Yaskawa INFORM job: DEMO_ROOF_SIDE_0625_3PAINT_53.JBI

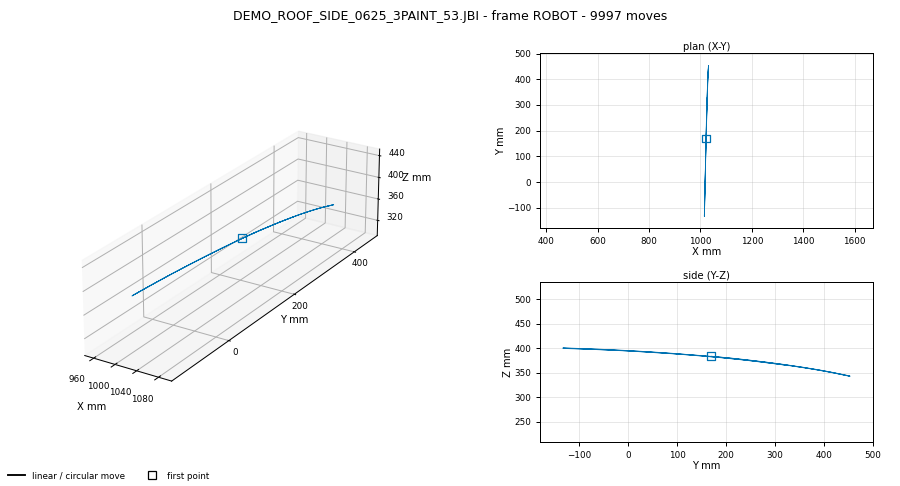
[picture p0: tool path of DEMO_ROOF_SIDE_0625_3PAINT_53.JBI in frame ROBOT, 9997 of 9997 moves have a stored position in this frame; points joined in program order, loops and branches not executed]
/JOB
//NAME DEMO_ROOF_SIDE_0625_3PAINT53
//POS
///NPOS 9997,0,0,0,0,0
///TOOL 0
///USER 0
///POSTYPE ROBOT
///RECTAN
///RCONF 1,0,0,0,0,0,0,0,0,0,0,0,0,0,0,0,0,0,0,0,0,0,0,0
C00000=1022.452,169.622,383.703,168.258,49.350,159.238
C00001=1022.457,169.870,383.681,168.261,49.345,159.237
C00002=1022.464,170.119,383.659,168.265,49.339,159.236
C00003=1022.469,170.368,383.637,168.268,49.333,159.236
C00004=1022.474,170.617,383.615,168.272,49.327,159.235
C00005=1022.480,170.866,383.593,168.276,49.321,159.234
C00006=1022.485,171.115,383.571,168.279,49.316,159.234
C00007=1022.491,171.398,383.546,168.283,49.310,159.233
C00008=1022.498,171.680,383.520,168.287,49.303,159.233
C00009=1022.504,171.963,383.496,168.291,49.296,159.232
C00010=1022.510,172.244,383.471,168.295,49.290,159.231
C00011=1022.515,172.494,383.449,168.299,49.284,159.231
C00012=1022.521,172.743,383.427,168.302,49.279,159.230
C00013=1022.526,172.991,383.404,168.306,49.273,159.229
C00014=1022.532,173.241,383.382,168.310,49.267,159.229
C00015=1022.537,173.489,383.361,168.313,49.261,159.228
C00016=1022.543,173.739,383.339,168.317,49.256,159.228
C00017=1022.548,173.988,383.316,168.320,49.250,159.227
C00018=1022.554,174.236,383.294,168.324,49.244,159.226
C00019=1022.559,174.486,383.272,168.328,49.238,159.226
C00020=1022.565,174.735,383.249,168.331,49.233,159.225
C00021=1022.571,174.983,383.228,168.335,49.227,159.225
C00022=1022.576,175.232,383.205,168.338,49.222,159.224
C00023=1022.582,175.481,383.183,168.342,49.216,159.223
C00024=1022.587,175.730,383.162,168.346,49.210,159.223
C00025=1022.593,175.979,383.139,168.349,49.204,159.222
C00026=1022.599,176.228,383.116,168.353,49.198,159.222
C00027=1022.603,176.477,383.094,168.357,49.193,159.221
C00028=1022.610,176.726,383.072,168.360,49.187,159.220
C00029=1022.615,176.975,383.050,168.364,49.181,159.220
C00030=1022.620,177.223,383.027,168.368,49.176,159.219
C00031=1022.627,177.473,383.006,168.372,49.170,159.219
C00032=1022.632,177.722,382.983,168.376,49.164,159.218
C00033=1022.637,177.970,382.961,168.379,49.159,159.217
C00034=1022.644,178.219,382.939,168.383,49.153,159.217
C00035=1022.649,178.469,382.916,168.387,49.147,159.216
C00036=1022.655,178.717,382.893,168.390,49.141,159.216
C00037=1022.660,178.966,382.871,168.394,49.136,159.215
C00038=1022.666,179.215,382.849,168.398,49.130,159.214
C00039=1022.671,179.464,382.827,168.401,49.125,159.214
C00040=1022.677,179.713,382.804,168.405,49.119,159.213
C00041=1022.683,179.962,382.783,168.409,49.113,159.213
C00042=1022.688,180.211,382.760,168.413,49.107,159.212
C00043=1022.694,180.460,382.738,168.416,49.102,159.211
C00044=1022.700,180.709,382.715,168.420,49.096,159.211
C00045=1022.706,180.958,382.693,168.424,49.090,159.210
C00046=1022.711,181.206,382.670,168.427,49.084,159.210
C00047=1022.717,181.455,382.647,168.432,49.079,159.209
C00048=1022.723,181.705,382.626,168.436,49.073,159.209
C00049=1022.729,181.953,382.603,168.440,49.067,159.208
C00050=1022.734,182.203,382.581,168.443,49.062,159.207
C00051=1022.740,182.452,382.558,168.447,49.056,159.207
C00052=1022.745,182.700,382.535,168.451,49.051,159.206
C00053=1022.750,182.949,382.512,168.454,49.045,159.206
C00054=1022.756,183.198,382.489,168.459,49.040,159.205
C00055=1022.761,183.448,382.466,168.462,49.034,159.205
C00056=1022.766,183.697,382.443,168.466,49.028,159.204
C00057=1022.771,183.945,382.420,168.470,49.023,159.204
C00058=1022.777,184.194,382.397,168.473,49.018,159.203
C00059=1022.782,184.443,382.374,168.478,49.013,159.203
C00060=1022.788,184.692,382.351,168.481,49.007,159.202
C00061=1022.793,184.941,382.328,168.485,49.002,159.201
C00062=1022.798,185.189,382.305,168.489,48.996,159.201
C00063=1022.803,185.438,382.282,168.492,48.991,159.200
C00064=1022.809,185.687,382.259,168.496,48.985,159.200
C00065=1022.814,185.936,382.235,168.501,48.980,159.199
C00066=1022.820,186.185,382.212,168.504,48.974,159.199
C00067=1022.826,186.434,382.189,168.508,48.969,159.198
C00068=1022.830,186.683,382.166,168.511,48.964,159.198
C00069=1022.836,186.932,382.143,168.515,48.958,159.197
C00070=1022.841,187.181,382.120,168.520,48.953,159.197
C00071=1022.848,187.462,382.094,168.524,48.947,159.196
C00072=1022.854,187.744,382.068,168.528,48.940,159.195
C00073=1022.860,188.026,382.041,168.532,48.934,159.195
C00074=1022.866,188.309,382.015,168.537,48.928,159.194
C00075=1022.871,188.558,381.992,168.541,48.922,159.194
C00076=1022.877,188.806,381.968,168.545,48.917,159.193
C00077=1022.882,189.055,381.945,168.549,48.911,159.193
C00078=1022.888,189.304,381.922,168.552,48.907,159.192
C00079=1022.894,189.553,381.899,168.556,48.901,159.191
C00080=1022.899,189.802,381.875,168.561,48.896,159.191
C00081=1022.905,190.051,381.852,168.564,48.890,159.190
C00082=1022.910,190.300,381.829,168.568,48.885,159.190
C00083=1022.916,190.548,381.805,168.572,48.879,159.189
C00084=1022.921,190.797,381.783,168.577,48.874,159.189
C00085=1022.926,191.046,381.759,168.580,48.868,159.188
C00086=1022.931,191.295,381.736,168.584,48.863,159.188
C00087=1022.937,191.543,381.712,168.588,48.857,159.187
C00088=1022.942,191.792,381.689,168.593,48.852,159.187
C00089=1022.948,192.041,381.666,168.596,48.847,159.186
C00090=1022.954,192.290,381.643,168.600,48.841,159.186
C00091=1022.959,192.539,381.619,168.604,48.836,159.185
C00092=1022.965,192.787,381.596,168.608,48.830,159.185
C00093=1022.971,193.036,381.573,168.611,48.825,159.184
C00094=1022.976,193.286,381.549,168.616,48.820,159.184
C00095=1022.982,193.534,381.526,168.620,48.814,159.183
C00096=1022.987,193.784,381.502,168.624,48.809,159.183
C00097=1022.993,194.033,381.479,168.628,48.803,159.182
C00098=1022.999,194.281,381.455,168.632,48.798,159.182
C00099=1023.004,194.530,381.432,168.636,48.792,159.181
C00100=1023.010,194.778,381.408,168.640,48.787,159.181
C00101=1023.016,195.027,381.385,168.644,48.781,159.180
C00102=1023.021,195.276,381.361,168.649,48.776,159.180
C00103=1023.027,195.525,381.338,168.653,48.770,159.179
C00104=1023.032,195.774,381.314,168.656,48.766,159.179
C00105=1023.038,196.023,381.291,168.660,48.760,159.178
C00106=1023.044,196.271,381.268,168.665,48.755,159.178
C00107=1023.049,196.520,381.244,168.669,48.749,159.177
C00108=1023.055,196.769,381.220,168.673,48.744,159.177
C00109=1023.061,197.018,381.197,168.677,48.738,159.176
C00110=1023.066,197.267,381.173,168.681,48.733,159.175
C00111=1023.072,197.516,381.150,168.685,48.727,159.175
C00112=1023.077,197.764,381.126,168.689,48.722,159.174
C00113=1023.083,198.013,381.103,168.693,48.716,159.174
C00114=1023.089,198.261,381.079,168.697,48.711,159.173
C00115=1023.095,198.511,381.055,168.702,48.706,159.173
C00116=1023.101,198.760,381.031,168.706,48.700,159.172
C00117=1023.106,199.009,381.008,168.710,48.695,159.172
C00118=1023.112,199.257,380.984,168.713,48.689,159.171
C00119=1023.117,199.506,380.961,168.718,48.684,159.171
C00120=1023.123,199.755,380.937,168.722,48.679,159.170
C00121=1023.129,200.004,380.913,168.726,48.673,159.170
C00122=1023.134,200.253,380.890,168.731,48.668,159.169
C00123=1023.140,200.501,380.865,168.735,48.663,159.169
C00124=1023.145,200.750,380.841,168.739,48.657,159.168
C00125=1023.151,200.999,380.816,168.743,48.653,159.168
C00126=1023.157,201.248,380.793,168.747,48.647,159.168
C00127=1023.162,201.497,380.769,168.751,48.642,159.167
C00128=1023.167,201.745,380.745,168.756,48.636,159.167
C00129=1023.173,201.994,380.721,168.760,48.631,159.166
C00130=1023.179,202.243,380.697,168.764,48.626,159.166
C00131=1023.184,202.492,380.672,168.769,48.621,159.165
C00132=1023.189,202.741,380.649,168.772,48.616,159.165
C00133=1023.195,202.989,380.625,168.776,48.610,159.164
C00134=1023.201,203.238,380.601,168.781,48.605,159.164
C00135=1023.225,204.270,380.500,169.200,48.703,159.246
C00136=1023.235,204.688,380.457,169.205,48.696,159.245
C00137=1023.246,205.107,380.414,169.211,48.689,159.244
C00138=1023.257,205.525,380.372,169.217,48.682,159.244
C00139=1023.268,205.943,380.328,169.222,48.674,159.243
C00140=1023.274,206.191,380.302,169.225,48.670,159.242
C00141=1023.281,206.440,380.277,169.228,48.666,159.242
C00142=1023.287,206.689,380.251,169.232,48.661,159.241
C00143=1023.294,206.937,380.225,169.234,48.657,159.241
C00144=1023.299,207.186,380.199,169.238,48.653,159.241
C00145=1023.306,207.434,380.173,169.241,48.648,159.240
C00146=1023.312,207.683,380.148,169.245,48.644,159.240
C00147=1023.319,207.932,380.121,169.248,48.640,159.239
C00148=1023.325,208.181,380.096,169.251,48.635,159.239
C00149=1023.332,208.429,380.070,169.255,48.631,159.238
C00150=1023.338,208.677,380.045,169.258,48.627,159.238
C00151=1023.345,208.926,380.018,169.261,48.623,159.238
C00152=1023.351,209.175,379.992,169.265,48.618,159.237
C00153=1023.357,209.423,379.966,169.267,48.615,159.237
C00154=1023.363,209.672,379.941,169.271,48.610,159.236
C00155=1023.371,209.920,379.914,169.275,48.606,159.236
C00156=1023.377,210.169,379.889,169.277,48.602,159.235
C00157=1023.383,210.417,379.862,169.281,48.598,159.235
C00158=1023.389,210.666,379.836,169.285,48.594,159.235
C00159=1023.396,210.915,379.811,169.287,48.590,159.234
C00160=1023.402,211.163,379.784,169.291,48.586,159.234
C00161=1023.408,211.411,379.758,169.295,48.581,159.234
C00162=1023.415,211.661,379.732,169.297,48.578,159.233
C00163=1023.421,211.909,379.706,169.301,48.573,159.233
C00164=1023.427,212.157,379.680,169.305,48.569,159.232
C00165=1023.433,212.406,379.654,169.307,48.565,159.232
C00166=1023.440,212.655,379.627,169.311,48.561,159.232
C00167=1023.446,212.903,379.601,169.315,48.557,159.231
C00168=1023.453,213.151,379.575,169.317,48.553,159.231
C00169=1023.459,213.401,379.549,169.321,48.549,159.230
C00170=1023.465,213.649,379.523,169.325,48.544,159.230
C00171=1023.471,213.897,379.496,169.327,48.541,159.230
C00172=1023.478,214.146,379.470,169.331,48.536,159.229
C00173=1023.485,214.394,379.444,169.335,48.532,159.229
C00174=1023.490,214.643,379.418,169.338,48.529,159.229
C00175=1023.497,214.892,379.391,169.341,48.524,159.228
C00176=1023.504,215.140,379.365,169.345,48.520,159.228
C00177=1023.510,215.389,379.339,169.348,48.516,159.227
C00178=1023.516,215.637,379.313,169.351,48.512,159.227
C00179=1023.523,215.885,379.287,169.355,48.508,159.227
C00180=1023.529,216.134,379.260,169.358,48.504,159.226
C00181=1023.536,216.382,379.234,169.362,48.500,159.226
C00182=1023.542,216.632,379.207,169.365,48.496,159.226
C00183=1023.549,216.880,379.181,169.368,48.492,159.225
C00184=1023.555,217.128,379.155,169.372,48.488,159.225
C00185=1023.561,217.377,379.128,169.375,48.484,159.224
C00186=1023.568,217.625,379.102,169.378,48.480,159.224
C00187=1023.575,217.874,379.076,169.382,48.476,159.224
C00188=1023.581,218.122,379.049,169.386,48.472,159.223
C00189=1023.587,218.371,379.023,169.388,48.468,159.223
C00190=1023.594,218.619,378.997,169.392,48.464,159.223
C00191=1023.600,218.868,378.970,169.396,48.460,159.222
C00192=1023.606,219.078,378.947,169.399,48.457,159.222
C00193=1023.611,219.289,378.925,169.401,48.454,159.222
C00194=1023.616,219.499,378.902,169.404,48.451,159.221
C00195=1023.622,219.710,378.879,169.407,48.447,159.221
C00196=1023.627,219.921,378.857,169.410,48.444,159.221
C00197=1023.632,220.131,378.834,169.413,48.441,159.221
C00198=1023.637,220.341,378.812,169.416,48.437,159.220
C00199=1023.643,220.552,378.789,169.419,48.434,159.220
C00200=1023.650,220.800,378.763,169.422,48.430,159.220
C00201=1023.656,221.049,378.736,169.425,48.426,159.219
C00202=1023.662,221.297,378.709,169.429,48.422,159.219
C00203=1023.669,221.546,378.683,169.432,48.419,159.219
C00204=1023.675,221.795,378.656,169.436,48.415,159.218
C00205=1023.681,222.044,378.629,169.439,48.411,159.218
C00206=1023.688,222.291,378.602,169.442,48.408,159.218
C00207=1023.694,222.540,378.575,169.446,48.404,159.217
C00208=1023.700,222.788,378.548,169.450,48.399,159.217
C00209=1023.707,223.037,378.522,169.453,48.396,159.217
C00210=1023.713,223.286,378.495,169.457,48.392,159.216
C00211=1023.719,223.534,378.468,169.459,48.388,159.216
C00212=1023.726,223.782,378.442,169.463,48.384,159.216
C00213=1023.732,224.031,378.415,169.467,48.381,159.215
C00214=1023.738,224.279,378.388,169.470,48.377,159.215
C00215=1023.746,224.528,378.361,169.474,48.373,159.215
C00216=1023.751,224.776,378.334,169.478,48.369,159.215
C00217=1023.758,225.025,378.307,169.480,48.366,159.214
C00218=1023.765,225.274,378.281,169.484,48.362,159.214
C00219=1023.771,225.522,378.253,169.488,48.358,159.214
C00220=1023.777,225.771,378.226,169.491,48.354,159.213
C00221=1023.784,226.019,378.200,169.495,48.351,159.213
C00222=1023.790,226.267,378.173,169.499,48.347,159.213
C00223=1023.797,226.516,378.146,169.501,48.343,159.212
C00224=1023.803,226.764,378.120,169.505,48.339,159.212
C00225=1023.810,227.013,378.092,169.508,48.336,159.212
C00226=1023.816,227.261,378.065,169.512,48.332,159.211
C00227=1023.822,227.509,378.037,169.516,48.328,159.211
C00228=1023.828,227.758,378.011,169.519,48.325,159.211
C00229=1023.835,228.007,377.984,169.523,48.321,159.210
C00230=1023.842,228.255,377.957,169.526,48.318,159.210
C00231=1023.848,228.503,377.930,169.530,48.314,159.210
C00232=1023.855,228.752,377.902,169.534,48.310,159.210
C00233=1023.861,229.001,377.875,169.537,48.307,159.209
C00234=1023.867,229.249,377.848,169.540,48.303,159.209
C00235=1023.874,229.497,377.820,169.544,48.299,159.209
C00236=1023.879,229.745,377.793,169.547,48.296,159.209
C00237=1023.886,229.994,377.766,169.551,48.292,159.208
C00238=1023.892,230.243,377.739,169.554,48.289,159.208
C00239=1023.899,230.491,377.711,169.558,48.285,159.208
C00240=1023.905,230.740,377.684,169.562,48.282,159.208
C00241=1023.912,230.988,377.657,169.565,48.278,159.207
C00242=1023.918,231.236,377.629,169.569,48.274,159.207
C00243=1023.924,231.485,377.602,169.572,48.271,159.207
C00244=1023.931,231.733,377.575,169.576,48.268,159.207
C00245=1023.937,231.981,377.547,169.580,48.264,159.206
C00246=1023.943,232.230,377.520,169.583,48.260,159.206
C00247=1023.950,232.479,377.492,169.587,48.257,159.206
C00248=1023.956,232.726,377.465,169.590,48.254,159.206
C00249=1023.963,232.975,377.437,169.594,48.250,159.205
C00250=1023.969,233.224,377.410,169.597,48.247,159.205
C00251=1023.975,233.473,377.382,169.601,48.243,159.205
C00252=1023.986,233.885,377.337,169.607,48.238,159.204
C00253=1023.997,234.298,377.291,169.612,48.232,159.204
C00254=1024.007,234.712,377.245,169.619,48.226,159.204
C00255=1024.017,235.125,377.199,169.625,48.220,159.203
C00256=1024.024,235.373,377.172,169.628,48.217,159.203
C00257=1024.031,235.621,377.144,169.632,48.213,159.203
C00258=1024.037,235.870,377.116,169.636,48.210,159.202
C00259=1024.043,236.118,377.089,169.639,48.207,159.202
C00260=1024.050,236.367,377.062,169.643,48.203,159.202
C00261=1024.056,236.615,377.034,169.646,48.199,159.202
C00262=1024.063,236.864,377.006,169.650,48.196,159.201
C00263=1024.069,237.112,376.978,169.654,48.193,159.201
C00264=1024.075,237.360,376.951,169.657,48.189,159.201
C00265=1024.082,237.609,376.923,169.661,48.186,159.201
C00266=1024.088,237.857,376.895,169.664,48.183,159.201
C00267=1024.095,238.105,376.868,169.668,48.179,159.200
C00268=1024.102,238.354,376.840,169.672,48.176,159.200
C00269=1024.108,238.603,376.811,169.675,48.173,159.200
C00270=1024.114,238.850,376.784,169.679,48.169,159.200
C00271=1024.120,239.099,376.756,169.684,48.166,159.200
C00272=1024.127,239.347,376.729,169.686,48.162,159.199
C00273=1024.134,239.596,376.701,169.690,48.159,159.199
C00274=1024.141,239.844,376.673,169.693,48.156,159.199
C00275=1024.146,240.092,376.645,169.698,48.153,159.199
C00276=1024.153,240.341,376.617,169.701,48.150,159.199
C00277=1024.158,240.589,376.589,169.705,48.146,159.198
C00278=1024.165,240.837,376.561,169.709,48.143,159.198
C00279=1024.171,241.086,376.532,169.712,48.140,159.198
C00280=1024.178,241.334,376.505,169.716,48.136,159.198
C00281=1024.185,241.583,376.477,169.719,48.133,159.198
C00282=1024.190,241.831,376.449,169.723,48.130,159.197
C00283=1024.197,242.079,376.421,169.727,48.126,159.197
C00284=1024.203,242.327,376.392,169.731,48.124,159.197
C00285=1024.210,242.576,376.364,169.735,48.121,159.197
C00286=1024.216,242.824,376.337,169.738,48.117,159.197
C00287=1024.223,243.072,376.308,169.742,48.114,159.197
C00288=1024.229,243.321,376.280,169.745,48.111,159.196
C00289=1024.235,243.570,376.252,169.749,48.107,159.196
C00290=1024.242,243.817,376.223,169.753,48.105,159.196
C00291=1024.248,244.065,376.195,169.757,48.102,159.196
C00292=1024.254,244.314,376.167,169.761,48.098,159.196
C00293=1024.261,244.562,376.138,169.764,48.095,159.195
C00294=1024.266,244.811,376.110,169.768,48.092,159.195
C00295=1024.273,245.059,376.081,169.771,48.089,159.195
C00296=1024.279,245.307,376.053,169.775,48.086,159.195
C00297=1024.286,245.556,376.024,169.779,48.083,159.195
C00298=1024.292,245.804,375.996,169.783,48.080,159.195
C00299=1024.299,246.052,375.968,169.787,48.077,159.195
C00300=1024.305,246.301,375.939,169.790,48.074,159.195
C00301=1024.311,246.549,375.910,169.794,48.071,159.194
C00302=1024.317,246.798,375.882,169.798,48.068,159.194
C00303=1024.324,247.046,375.853,169.802,48.065,159.194
C00304=1024.330,247.294,375.825,169.805,48.062,159.194
C00305=1024.336,247.542,375.796,169.809,48.059,159.194
C00306=1024.343,247.791,375.768,169.812,48.056,159.194
C00307=1024.349,248.039,375.739,169.817,48.053,159.194
C00308=1024.359,248.446,375.693,169.823,48.047,159.193
C00309=1024.370,248.853,375.646,169.829,48.043,159.193
C00310=1024.380,249.260,375.599,169.836,48.038,159.193
C00311=1024.390,249.666,375.551,169.841,48.033,159.193
C00312=1024.397,249.915,375.524,169.845,48.030,159.193
C00313=1024.403,250.163,375.495,169.849,48.027,159.192
C00314=1024.409,250.411,375.466,169.853,48.024,159.192
C00315=1024.416,250.660,375.438,169.856,48.021,159.192
C00316=1024.422,250.908,375.409,169.860,48.018,159.192
C00317=1024.429,251.156,375.380,169.865,48.015,159.192
C00318=1024.435,251.404,375.351,169.868,48.012,159.192
C00319=1024.442,251.652,375.323,169.872,48.009,159.192
C00320=1024.448,251.901,375.294,169.875,48.006,159.192
C00321=1024.454,252.149,375.265,169.880,48.004,159.192
C00322=1024.461,252.396,375.236,169.884,48.000,159.191
C00323=1024.468,252.646,375.208,169.887,47.998,159.191
C00324=1024.474,252.894,375.179,169.892,47.995,159.191
C00325=1024.480,253.142,375.150,169.895,47.992,159.191
C00326=1024.487,253.390,375.121,169.899,47.989,159.191
C00327=1024.493,253.638,375.092,169.903,47.986,159.191
C00328=1024.499,253.887,375.064,169.907,47.983,159.191
C00329=1024.506,254.135,375.035,169.911,47.980,159.191
C00330=1024.513,254.384,375.006,169.914,47.977,159.191
C00331=1024.519,254.632,374.977,169.918,47.975,159.191
C00332=1024.526,254.880,374.948,169.922,47.971,159.190
C00333=1024.533,255.128,374.920,169.926,47.969,159.190
C00334=1024.539,255.376,374.890,169.930,47.966,159.190
C00335=1024.546,255.625,374.861,169.934,47.963,159.190
C00336=1024.552,255.873,374.833,169.938,47.960,159.190
C00337=1024.559,256.121,374.804,169.942,47.957,159.190
C00338=1024.565,256.369,374.775,169.945,47.954,159.190
C00339=1024.571,256.617,374.746,169.950,47.952,159.190
C00340=1024.578,256.866,374.717,169.954,47.948,159.190
C00341=1024.585,257.114,374.688,169.957,47.946,159.189
C00342=1024.591,257.362,374.659,169.961,47.943,159.190
C00343=1024.597,257.610,374.630,169.966,47.940,159.190
C00344=1024.604,257.859,374.601,169.969,47.937,159.189
C00345=1024.611,258.107,374.572,169.973,47.934,159.189
C00346=1024.618,258.355,374.543,169.978,47.932,159.189
C00347=1024.624,258.604,374.514,169.981,47.929,159.189
C00348=1024.631,258.852,374.485,169.985,47.926,159.189
C00349=1024.638,259.100,374.456,169.990,47.923,159.189
C00350=1024.645,259.348,374.426,169.993,47.921,159.189
C00351=1024.651,259.596,374.397,169.997,47.917,159.189
C00352=1024.657,259.844,374.368,170.001,47.915,159.189
C00353=1024.665,260.093,374.339,170.005,47.912,159.189
C00354=1024.671,260.341,374.310,170.009,47.909,159.189
C00355=1024.677,260.589,374.281,170.014,47.907,159.189
C00356=1024.684,260.837,374.252,170.017,47.904,159.189
C00357=1024.691,261.086,374.222,170.022,47.901,159.189
C00358=1024.697,261.334,374.193,170.025,47.899,159.188
C00359=1024.703,261.582,374.164,170.029,47.896,159.188
C00360=1024.710,261.830,374.134,170.034,47.894,159.188
C00361=1024.716,262.078,374.104,170.037,47.891,159.188
C00362=1024.722,262.326,374.075,170.042,47.888,159.188
C00363=1024.729,262.575,374.045,170.045,47.886,159.188
C00364=1024.739,262.980,373.997,170.052,47.881,159.188
C00365=1024.750,263.385,373.948,170.058,47.877,159.188
C00366=1024.760,263.791,373.901,170.065,47.873,159.188
C00367=1024.772,264.196,373.852,170.072,47.869,159.188
C00368=1024.778,264.444,373.823,170.075,47.866,159.188
C00369=1024.785,264.692,373.793,170.080,47.863,159.188
C00370=1024.791,264.941,373.764,170.083,47.861,159.188
C00371=1024.798,265.189,373.733,170.088,47.858,159.188
C00372=1024.804,265.437,373.704,170.092,47.856,159.188
C00373=1024.811,265.684,373.675,170.095,47.853,159.188
C00374=1024.817,265.934,373.645,170.100,47.851,159.188
C00375=1024.824,266.181,373.615,170.105,47.848,159.188
C00376=1024.831,266.429,373.585,170.108,47.846,159.188
C00377=1024.836,266.678,373.555,170.112,47.843,159.188
C00378=1024.843,266.925,373.525,170.116,47.841,159.188
C00379=1024.850,267.173,373.495,170.120,47.839,159.188
C00380=1024.856,267.422,373.466,170.125,47.836,159.188
C00381=1024.863,267.670,373.435,170.128,47.833,159.188
C00382=1024.869,267.918,373.406,170.133,47.831,159.188
C00383=1024.876,268.166,373.376,170.137,47.829,159.188
C00384=1024.882,268.414,373.346,170.141,47.826,159.188
C00385=1024.889,268.662,373.316,170.145,47.823,159.188
C00386=1024.896,268.910,373.286,170.149,47.821,159.188
C00387=1024.902,269.159,373.256,170.153,47.819,159.188
C00388=1024.908,269.407,373.226,170.158,47.816,159.188
C00389=1024.915,269.655,373.196,170.161,47.814,159.188
C00390=1024.921,269.903,373.166,170.166,47.812,159.188
C00391=1024.928,270.151,373.136,170.170,47.809,159.188
C00392=1024.934,270.399,373.105,170.174,47.806,159.188
C00393=1024.941,270.647,373.075,170.178,47.804,159.188
C00394=1024.947,270.895,373.045,170.183,47.802,159.188
C00395=1024.954,271.144,373.015,170.186,47.800,159.189
C00396=1024.960,271.391,372.985,170.191,47.797,159.189
C00397=1024.967,271.640,372.955,170.195,47.795,159.189
C00398=1024.974,271.887,372.925,170.199,47.793,159.189
C00399=1024.980,272.136,372.895,170.204,47.791,159.189
C00400=1024.987,272.384,372.864,170.207,47.788,159.189
C00401=1024.993,272.632,372.834,170.212,47.785,159.189
C00402=1025.000,272.880,372.804,170.216,47.783,159.189
C00403=1025.006,273.128,372.774,170.220,47.781,159.189
C00404=1025.013,273.376,372.743,170.224,47.779,159.189
C00405=1025.020,273.624,372.712,170.229,47.777,159.189
C00406=1025.026,273.872,372.682,170.233,47.774,159.189
C00407=1025.033,274.120,372.652,170.237,47.772,159.189
C00408=1025.039,274.368,372.621,170.242,47.770,159.189
C00409=1025.046,274.616,372.591,170.245,47.768,159.189
C00410=1025.052,274.864,372.560,170.250,47.765,159.189
C00411=1025.058,275.112,372.530,170.255,47.763,159.189
C00412=1025.065,275.360,372.500,170.258,47.761,159.190
C00413=1025.072,275.608,372.468,170.263,47.758,159.190
C00414=1025.078,275.856,372.439,170.267,47.756,159.190
C00415=1025.085,276.104,372.408,170.271,47.754,159.190
C00416=1025.092,276.353,372.378,170.275,47.752,159.190
C00417=1025.098,276.600,372.347,170.280,47.750,159.190
C00418=1025.104,276.848,372.316,170.284,47.747,159.190
C00419=1025.112,277.097,372.286,170.288,47.745,159.190
C00420=1025.122,277.507,372.235,170.296,47.742,159.190
C00421=1025.132,277.916,372.184,170.302,47.738,159.190
C00422=1025.143,278.326,372.133,170.310,47.735,159.191
C00423=1025.154,278.736,372.083,170.317,47.731,159.191
C00424=1025.161,278.984,372.052,170.321,47.729,159.191
C00425=1025.168,279.232,372.020,170.326,47.727,159.191
C00426=1025.174,279.481,371.990,170.330,47.725,159.191
C00427=1025.180,279.728,371.959,170.334,47.723,159.191
C00428=1025.187,279.977,371.928,170.338,47.721,159.191
C00429=1025.194,280.224,371.897,170.343,47.719,159.192
C00430=1025.200,280.473,371.866,170.347,47.717,159.192
C00431=1025.207,280.720,371.835,170.352,47.715,159.192
C00432=1025.213,280.968,371.805,170.356,47.713,159.192
C00433=1025.220,281.216,371.773,170.360,47.711,159.192
C00434=1025.226,281.464,371.742,170.365,47.709,159.192
C00435=1025.234,281.712,371.712,170.369,47.706,159.192
C00436=1025.240,281.960,371.681,170.373,47.704,159.192
C00437=1025.246,282.208,371.650,170.378,47.702,159.193
C00438=1025.253,282.456,371.618,170.382,47.700,159.193
C00439=1025.260,282.704,371.587,170.387,47.698,159.193
C00440=1025.266,282.952,371.556,170.391,47.696,159.193
C00441=1025.273,283.200,371.525,170.395,47.694,159.193
C00442=1025.280,283.447,371.494,170.400,47.692,159.193
C00443=1025.286,283.696,371.464,170.404,47.691,159.193
C00444=1025.293,283.944,371.432,170.409,47.688,159.194
C00445=1025.299,284.192,371.401,170.413,47.686,159.194
C00446=1025.306,284.439,371.369,170.418,47.684,159.194
C00447=1025.313,284.688,371.339,170.422,47.683,159.194
C00448=1025.320,284.936,371.308,170.427,47.680,159.194
C00449=1025.327,285.183,371.276,170.431,47.678,159.194
C00450=1025.333,285.431,371.245,170.435,47.677,159.194
C00451=1025.340,285.679,371.213,170.440,47.675,159.195
C00452=1025.346,285.926,371.182,170.445,47.673,159.195
C00453=1025.353,286.174,371.151,170.449,47.671,159.195
C00454=1025.359,286.423,371.120,170.453,47.669,159.195
C00455=1025.366,286.671,371.089,170.458,47.667,159.195
C00456=1025.373,286.919,371.057,170.463,47.665,159.196
C00457=1025.379,287.167,371.025,170.467,47.664,159.196
C00458=1025.386,287.415,370.994,170.471,47.662,159.196
C00459=1025.392,287.663,370.962,170.476,47.660,159.196
C00460=1025.399,287.911,370.931,170.481,47.658,159.196
C00461=1025.406,288.159,370.900,170.485,47.657,159.197
C00462=1025.413,288.406,370.867,170.490,47.655,159.197
C00463=1025.420,288.654,370.836,170.494,47.653,159.197
C00464=1025.426,288.902,370.805,170.498,47.651,159.197
C00465=1025.433,289.150,370.773,170.503,47.649,159.197
C00466=1025.439,289.398,370.741,170.508,47.647,159.198
C00467=1025.446,289.646,370.710,170.513,47.645,159.198
C00468=1025.452,289.894,370.678,170.517,47.644,159.198
C00469=1025.459,290.141,370.647,170.521,47.642,159.198
C00470=1025.466,290.389,370.615,170.526,47.640,159.198
C00471=1025.473,290.637,370.583,170.531,47.638,159.199
C00472=1025.479,290.885,370.551,170.535,47.637,159.199
C00473=1025.486,291.133,370.520,170.540,47.635,159.199
C00474=1025.493,291.380,370.488,170.545,47.633,159.199
C00475=1025.500,291.629,370.456,170.549,47.631,159.199
C00476=1025.505,291.839,370.429,170.553,47.630,159.200
C00477=1025.511,292.051,370.402,170.557,47.628,159.200
C00478=1025.516,292.261,370.375,170.561,47.627,159.200
C00479=1025.523,292.472,370.348,170.565,47.626,159.200
C00480=1025.528,292.684,370.321,170.569,47.624,159.200
C00481=1025.533,292.895,370.293,170.573,47.623,159.201
C00482=1025.540,293.106,370.266,170.577,47.621,159.201
C00483=1025.545,293.317,370.238,170.581,47.620,159.201
C00484=1025.552,293.565,370.207,170.585,47.618,159.201
C00485=1025.559,293.813,370.175,170.590,47.617,159.202
C00486=1025.565,294.061,370.143,170.594,47.615,159.202
C00487=1025.572,294.308,370.111,170.599,47.613,159.202
C00488=1025.578,294.556,370.079,170.604,47.612,159.202
C00489=1025.585,294.804,370.046,170.609,47.611,159.203
C00490=1025.592,295.051,370.014,170.613,47.609,159.203
C00491=1025.598,295.300,369.981,170.618,47.607,159.203
C00492=1025.604,295.548,369.948,170.623,47.606,159.204
C00493=1025.611,295.795,369.916,170.627,47.605,159.204
C00494=1025.617,296.043,369.884,170.632,47.603,159.204
C00495=1025.624,296.290,369.852,170.637,47.601,159.204
C00496=1025.631,296.538,369.819,170.642,47.600,159.205
C00497=1025.637,296.787,369.787,170.646,47.599,159.205
C00498=1025.644,297.034,369.755,170.651,47.597,159.205
C00499=1025.651,297.282,369.722,170.656,47.595,159.206
C00500=1025.657,297.529,369.689,170.661,47.594,159.206
C00501=1025.664,297.777,369.657,170.666,47.592,159.206
C00502=1025.671,298.026,369.625,170.670,47.591,159.206
C00503=1025.677,298.273,369.592,170.675,47.590,159.207
C00504=1025.684,298.520,369.560,170.680,47.588,159.207
C00505=1025.690,298.768,369.527,170.685,47.586,159.207
C00506=1025.698,299.016,369.495,170.689,47.585,159.208
C00507=1025.704,299.264,369.462,170.694,47.584,159.208
C00508=1025.710,299.511,369.429,170.699,47.582,159.208
C00509=1025.717,299.759,369.398,170.704,47.581,159.209
C00510=1025.724,300.007,369.365,170.709,47.580,159.209
C00511=1025.730,300.255,369.332,170.713,47.578,159.209
C00512=1025.737,300.502,369.300,170.718,47.577,159.210
C00513=1025.744,300.751,369.267,170.723,47.576,159.210
C00514=1025.751,300.998,369.234,170.728,47.574,159.210
C00515=1025.758,301.245,369.202,170.733,47.573,159.211
C00516=1025.764,301.494,369.169,170.737,47.572,159.211
C00517=1025.771,301.741,369.136,170.742,47.570,159.211
C00518=1025.778,301.989,369.103,170.747,47.569,159.212
C00519=1025.785,302.236,369.070,170.752,47.567,159.212
C00520=1025.791,302.484,369.037,170.757,47.566,159.212
C00521=1025.799,302.732,369.005,170.762,47.564,159.213
C00522=1025.805,302.979,368.972,170.767,47.563,159.213
C00523=1025.812,303.228,368.939,170.771,47.562,159.213
C00524=1025.819,303.475,368.907,170.776,47.560,159.214
C00525=1025.825,303.723,368.874,170.781,47.559,159.214
C00526=1025.832,303.971,368.841,170.786,47.558,159.214
C00527=1025.840,304.218,368.808,170.791,47.556,159.215
C00528=1025.847,304.466,368.775,170.797,47.555,159.215
C00529=1025.853,304.713,368.742,170.802,47.554,159.215
C00530=1025.861,304.961,368.710,170.806,47.553,159.216
C00531=1025.867,305.208,368.676,170.811,47.551,159.216
C00532=1025.874,305.457,368.643,170.816,47.550,159.216
C00533=1025.881,305.704,368.611,170.821,47.549,159.217
C00534=1025.888,305.952,368.578,170.826,47.547,159.217
C00535=1025.895,306.200,368.544,170.831,47.546,159.218
C00536=1025.901,306.419,368.515,170.835,47.545,159.218
C00537=1025.907,306.639,368.486,170.840,47.544,159.218
C00538=1025.914,306.859,368.457,170.845,47.543,159.219
C00539=1025.920,307.078,368.427,170.849,47.542,159.219
C00540=1025.926,307.298,368.398,170.854,47.541,159.219
C00541=1025.933,307.518,368.368,170.858,47.540,159.220
C00542=1025.939,307.738,368.339,170.862,47.538,159.220
C00543=1025.945,307.958,368.310,170.867,47.537,159.220
C00544=1025.952,308.205,368.277,170.872,47.536,159.221
C00545=1025.959,308.453,368.243,170.877,47.535,159.221
C00546=1025.966,308.700,368.211,170.882,47.533,159.221
C00547=1025.973,308.948,368.177,170.888,47.533,159.222
C00548=1025.980,309.196,368.144,170.892,47.531,159.222
C00549=1025.987,309.443,368.111,170.897,47.530,159.223
C00550=1025.994,309.691,368.078,170.902,47.529,159.223
C00551=1026.001,309.939,368.044,170.907,47.528,159.223
C00552=1026.008,310.186,368.012,170.912,47.526,159.224
C00553=1026.016,310.434,367.979,170.918,47.526,159.224
C00554=1026.023,310.681,367.945,170.923,47.524,159.225
C00555=1026.029,310.929,367.912,170.928,47.523,159.225
C00556=1026.036,311.177,367.878,170.933,47.522,159.226
C00557=1026.043,311.425,367.844,170.938,47.521,159.226
C00558=1026.049,311.672,367.810,170.944,47.520,159.227
C00559=1026.057,311.919,367.776,170.949,47.519,159.227
C00560=1026.063,312.167,367.742,170.954,47.518,159.227
C00561=1026.070,312.414,367.709,170.959,47.518,159.228
C00562=1026.077,312.662,367.675,170.964,47.517,159.228
C00563=1026.083,312.910,367.640,170.969,47.515,159.229
C00564=1026.090,313.157,367.607,170.974,47.515,159.229
C00565=1026.097,313.405,367.573,170.980,47.514,159.230
C00566=1026.104,313.653,367.539,170.985,47.512,159.230
C00567=1026.111,313.900,367.505,170.990,47.512,159.231
C00568=1026.117,314.147,367.471,170.995,47.511,159.231
C00569=1026.125,314.395,367.437,171.001,47.510,159.232
C00570=1026.131,314.643,367.403,171.006,47.509,159.232
C00571=1026.138,314.891,367.369,171.011,47.508,159.233
C00572=1026.145,315.138,367.336,171.017,47.507,159.233
C00573=1026.152,315.385,367.301,171.022,47.506,159.234
C00574=1026.159,315.633,367.267,171.026,47.506,159.234
C00575=1026.166,315.880,367.233,171.032,47.505,159.235
C00576=1026.173,316.128,367.199,171.037,47.504,159.235
C00577=1026.180,316.376,367.165,171.042,47.503,159.236
C00578=1026.186,316.623,367.131,171.048,47.503,159.236
C00579=1026.193,316.870,367.096,171.053,47.501,159.236
C00580=1026.200,317.118,367.062,171.058,47.500,159.237
C00581=1026.208,317.366,367.029,171.063,47.500,159.238
C00582=1026.214,317.613,366.993,171.069,47.499,159.238
C00583=1026.221,317.861,366.960,171.074,47.498,159.239
C00584=1026.229,318.108,366.926,171.079,47.497,159.239
C00585=1026.235,318.356,366.891,171.085,47.496,159.240
C00586=1026.243,318.603,366.857,171.090,47.496,159.240
C00587=1026.250,318.851,366.823,171.096,47.495,159.241
C00588=1026.257,319.098,366.788,171.101,47.494,159.241
C00589=1026.264,319.346,366.754,171.106,47.493,159.242
C00590=1026.271,319.594,366.720,171.112,47.492,159.242
C00591=1026.278,319.841,366.685,171.117,47.492,159.243
C00592=1026.285,320.089,366.651,171.123,47.491,159.243
C00593=1026.293,320.336,366.617,171.129,47.490,159.244
C00594=1026.299,320.584,366.582,171.134,47.490,159.245
C00595=1026.306,320.831,366.548,171.140,47.489,159.245
C00596=1026.312,321.053,366.517,171.144,47.488,159.246
C00597=1026.319,321.276,366.486,171.149,47.487,159.246
C00598=1026.325,321.498,366.455,171.154,47.487,159.247
C00599=1026.332,321.720,366.425,171.159,47.486,159.247
C00600=1026.339,321.942,366.393,171.163,47.486,159.247
C00601=1026.345,322.164,366.362,171.169,47.485,159.248
C00602=1026.351,322.387,366.331,171.173,47.484,159.248
C00603=1026.358,322.609,366.300,171.178,47.484,159.249
C00604=1026.365,322.856,366.266,171.184,47.483,159.250
C00605=1026.371,323.104,366.231,171.189,47.483,159.250
C00606=1026.380,323.352,366.196,171.195,47.482,159.251
C00607=1026.387,323.599,366.162,171.200,47.481,159.251
C00608=1026.394,323.846,366.127,171.207,47.480,159.252
C00609=1026.401,324.094,366.093,171.212,47.480,159.253
C00610=1026.409,324.341,366.058,171.218,47.479,159.253
C00611=1026.416,324.589,366.023,171.223,47.479,159.254
C00612=1026.423,324.836,365.988,171.229,47.478,159.254
C00613=1026.430,325.084,365.954,171.234,47.477,159.255
C00614=1026.437,325.331,365.919,171.240,47.477,159.256
C00615=1026.446,325.579,365.884,171.245,47.476,159.256
C00616=1026.452,325.826,365.849,171.251,47.475,159.257
C00617=1026.460,326.073,365.815,171.257,47.475,159.257
C00618=1026.468,326.321,365.780,171.262,47.474,159.258
C00619=1026.475,326.568,365.745,171.268,47.474,159.259
C00620=1026.482,326.816,365.711,171.273,47.473,159.259
C00621=1026.489,327.064,365.675,171.279,47.472,159.260
C00622=1026.497,327.311,365.641,171.285,47.472,159.260
C00623=1026.504,327.558,365.605,171.291,47.472,159.261
C00624=1026.512,327.806,365.570,171.296,47.471,159.262
C00625=1026.519,328.053,365.535,171.302,47.471,159.262
C00626=1026.525,328.300,365.500,171.308,47.471,159.263
C00627=1026.532,328.548,365.465,171.313,47.470,159.264
C00628=1026.540,328.795,365.428,171.319,47.470,159.264
C00629=1026.547,329.042,365.394,171.325,47.469,159.265
C00630=1026.555,329.290,365.358,171.331,47.468,159.265
C00631=1026.562,329.538,365.323,171.336,47.468,159.266
C00632=1026.569,329.785,365.287,171.342,47.468,159.267
C00633=1026.576,330.033,365.252,171.348,47.468,159.268
C00634=1026.583,330.280,365.217,171.353,47.467,159.268
C00635=1026.591,330.527,365.181,171.360,47.466,159.269
C00636=1026.598,330.774,365.146,171.365,47.466,159.270
C00637=1026.605,331.022,365.111,171.371,47.466,159.270
C00638=1026.612,331.269,365.075,171.377,47.466,159.271
C00639=1026.619,331.517,365.039,171.382,47.466,159.272
C00640=1026.627,331.764,365.003,171.389,47.465,159.272
C00641=1026.634,332.011,364.969,171.394,47.464,159.273
C00642=1026.642,332.259,364.932,171.400,47.464,159.274
C00643=1026.649,332.506,364.897,171.406,47.464,159.274
C00644=1026.656,332.753,364.861,171.411,47.464,159.275
C00645=1026.663,333.001,364.826,171.418,47.463,159.276
C00646=1026.671,333.248,364.790,171.424,47.463,159.277
C00647=1026.679,333.496,364.755,171.430,47.463,159.277
C00648=1026.686,333.743,364.719,171.435,47.463,159.278
C00649=1026.694,333.990,364.683,171.442,47.462,159.279
C00650=1026.701,334.237,364.647,171.448,47.462,159.279
C00651=1026.708,334.485,364.611,171.453,47.462,159.280
C00652=1026.715,334.732,364.575,171.459,47.462,159.281
C00653=1026.722,334.979,364.539,171.466,47.461,159.282
C00654=1026.730,335.227,364.503,171.472,47.462,159.283
C00655=1026.737,335.474,364.467,171.477,47.462,159.283
C00656=1026.744,335.694,364.436,171.483,47.462,159.284
C00657=1026.750,335.914,364.403,171.488,47.462,159.285
C00658=1026.757,336.134,364.371,171.493,47.461,159.285
C00659=1026.763,336.354,364.339,171.499,47.461,159.286
C00660=1026.770,336.574,364.307,171.505,47.461,159.287
C00661=1026.776,336.794,364.275,171.509,47.461,159.287
C00662=1026.783,337.014,364.242,171.515,47.461,159.288
C00663=1026.790,337.234,364.210,171.520,47.461,159.289
C00664=1026.797,337.481,364.174,171.526,47.461,159.289
C00665=1026.804,337.729,364.138,171.532,47.460,159.290
C00666=1026.812,337.976,364.102,171.539,47.461,159.291
C00667=1026.820,338.224,364.065,171.544,47.460,159.292
C00668=1026.827,338.470,364.029,171.550,47.460,159.292
C00669=1026.834,338.718,363.993,171.557,47.460,159.293
C00670=1026.842,338.965,363.957,171.563,47.460,159.294
C00671=1026.850,339.213,363.921,171.568,47.460,159.295
C00672=1026.857,339.459,363.884,171.575,47.460,159.296
C00673=1026.865,339.706,363.848,171.581,47.460,159.297
C00674=1026.872,339.954,363.812,171.587,47.460,159.297
C00675=1026.879,340.201,363.775,171.594,47.460,159.298
C00676=1026.887,340.448,363.738,171.600,47.460,159.299
C00677=1026.895,340.696,363.702,171.605,47.460,159.300
C00678=1026.901,340.943,363.665,171.612,47.460,159.301
C00679=1026.909,341.190,363.628,171.618,47.460,159.301
C00680=1026.917,341.437,363.592,171.624,47.460,159.302
C00681=1026.924,341.685,363.555,171.631,47.461,159.303
C00682=1026.932,341.932,363.519,171.637,47.460,159.304
C00683=1026.940,342.179,363.482,171.643,47.461,159.305
C00684=1026.947,342.426,363.445,171.650,47.461,159.306
C00685=1026.955,342.674,363.409,171.655,47.461,159.307
C00686=1026.963,342.921,363.372,171.662,47.461,159.307
C00687=1026.969,343.168,363.335,171.668,47.461,159.308
C00688=1026.977,343.415,363.298,171.674,47.462,159.309
C00689=1026.984,343.662,363.261,171.681,47.461,159.310
C00690=1026.992,343.909,363.224,171.687,47.462,159.311
C00691=1027.000,344.156,363.188,171.694,47.462,159.312
C00692=1027.007,344.404,363.151,171.700,47.462,159.313
C00693=1027.015,344.650,363.114,171.707,47.462,159.314
C00694=1027.022,344.898,363.076,171.713,47.463,159.315
C00695=1027.030,345.145,363.039,171.719,47.463,159.315
C00696=1027.037,345.393,363.002,171.726,47.463,159.316
C00697=1027.045,345.640,362.965,171.732,47.463,159.317
C00698=1027.053,345.886,362.928,171.739,47.463,159.318
C00699=1027.061,346.134,362.891,171.745,47.464,159.319
C00700=1027.069,346.380,362.854,171.752,47.464,159.320
C00701=1027.076,346.628,362.816,171.758,47.464,159.321
C00702=1027.084,346.875,362.780,171.764,47.464,159.322
C00703=1027.091,347.122,362.743,171.770,47.465,159.323
C00704=1027.099,347.369,362.706,171.777,47.465,159.324
C00705=1027.107,347.617,362.668,171.783,47.465,159.325
C00706=1027.115,347.864,362.631,171.791,47.466,159.326
C00707=1027.122,348.111,362.593,171.797,47.466,159.327
C00708=1027.130,348.358,362.556,171.804,47.467,159.327
C00709=1027.137,348.605,362.519,171.810,47.467,159.328
C00710=1027.146,348.852,362.481,171.817,47.467,159.329
C00711=1027.153,349.099,362.443,171.823,47.468,159.330
C00712=1027.160,349.346,362.406,171.830,47.468,159.331
C00713=1027.168,349.593,362.369,171.836,47.469,159.332
C00714=1027.176,349.840,362.331,171.843,47.469,159.333
C00715=1027.184,350.087,362.293,171.849,47.470,159.334
C00716=1027.190,350.305,362.259,171.855,47.470,159.335
C00717=1027.197,350.524,362.227,171.861,47.470,159.336
C00718=1027.204,350.742,362.193,171.867,47.470,159.337
C00719=1027.211,350.961,362.160,171.873,47.471,159.338
C00720=1027.218,351.180,362.126,171.879,47.471,159.339
C00721=1027.225,351.397,362.093,171.885,47.472,159.339
C00722=1027.231,351.616,362.060,171.891,47.472,159.340
C00723=1027.238,351.834,362.026,171.897,47.473,159.341
C00724=1027.245,352.081,361.989,171.903,47.473,159.342
C00725=1027.254,352.328,361.951,171.910,47.474,159.343
C00726=1027.262,352.576,361.913,171.917,47.474,159.344
C00727=1027.270,352.823,361.875,171.923,47.475,159.345
C00728=1027.278,353.070,361.838,171.931,47.475,159.346
C00729=1027.285,353.316,361.799,171.938,47.476,159.348
C00730=1027.293,353.564,361.761,171.944,47.477,159.348
C00731=1027.301,353.810,361.723,171.951,47.477,159.350
C00732=1027.310,354.057,361.685,171.957,47.478,159.350
C00733=1027.317,354.304,361.648,171.965,47.478,159.352
C00734=1027.325,354.552,361.609,171.972,47.479,159.353
C00735=1027.333,354.798,361.571,171.978,47.480,159.354
C00736=1027.341,355.046,361.534,171.985,47.480,159.355
C00737=1027.349,355.292,361.495,171.993,47.481,159.356
C00738=1027.357,355.539,361.457,171.999,47.482,159.357
C00739=1027.364,355.786,361.418,172.006,47.482,159.358
C00740=1027.373,356.033,361.380,172.013,47.483,159.359
C00741=1027.380,356.280,361.342,172.020,47.484,159.360
C00742=1027.388,356.527,361.303,172.027,47.485,159.361
C00743=1027.396,356.773,361.265,172.034,47.485,159.362
C00744=1027.404,357.021,361.226,172.041,47.486,159.364
C00745=1027.412,357.268,361.187,172.048,47.487,159.365
C00746=1027.420,357.514,361.149,172.055,47.487,159.366
C00747=1027.428,357.762,361.111,172.062,47.488,159.367
C00748=1027.437,358.009,361.073,172.069,47.489,159.368
C00749=1027.444,358.255,361.034,172.076,47.490,159.369
C00750=1027.452,358.502,360.996,172.083,47.490,159.370
C00751=1027.461,358.749,360.957,172.090,47.491,159.371
C00752=1027.468,358.996,360.919,172.097,47.492,159.372
C00753=1027.477,359.243,360.880,172.104,47.493,159.374
C00754=1027.485,359.490,360.841,172.111,47.494,159.375
C00755=1027.492,359.736,360.803,172.119,47.495,159.376
C00756=1027.500,359.984,360.764,172.126,47.495,159.377
C00757=1027.509,360.230,360.725,172.133,47.496,159.378
C00758=1027.517,360.477,360.686,172.140,47.497,159.379
C00759=1027.525,360.724,360.648,172.147,47.498,159.381
C00760=1027.532,360.971,360.608,172.155,47.499,159.382
C00761=1027.540,361.218,360.569,172.162,47.500,159.383
C00762=1027.549,361.465,360.530,172.170,47.501,159.384
C00763=1027.557,361.712,360.491,172.177,47.502,159.385
C00764=1027.564,361.958,360.452,172.183,47.503,159.387
C00765=1027.573,362.205,360.413,172.191,47.504,159.388
C00766=1027.581,362.452,360.374,172.198,47.505,159.389
C00767=1027.589,362.698,360.335,172.206,47.506,159.390
C00768=1027.597,362.945,360.295,172.213,47.507,159.392
C00769=1027.605,363.193,360.256,172.221,47.508,159.393
C00770=1027.613,363.438,360.217,172.228,47.509,159.394
C00771=1027.621,363.685,360.178,172.235,47.510,159.395
C00772=1027.629,363.932,360.138,172.242,47.511,159.396
C00773=1027.637,364.179,360.099,172.250,47.512,159.398
C00774=1027.646,364.426,360.060,172.257,47.513,159.399
C00775=1027.654,364.672,360.021,172.264,47.514,159.400
C00776=1027.661,364.894,359.985,172.271,47.515,159.401
C00777=1027.669,365.116,359.949,172.278,47.516,159.402
C00778=1027.676,365.338,359.915,172.284,47.517,159.404
C00779=1027.683,365.559,359.879,172.291,47.519,159.405
C00780=1027.691,365.780,359.843,172.298,47.519,159.406
C00781=1027.699,366.003,359.808,172.305,47.520,159.407
C00782=1027.706,366.224,359.772,172.312,47.521,159.408
C00783=1027.713,366.446,359.737,172.319,47.523,159.409
C00784=1027.721,366.693,359.697,172.326,47.524,159.411
C00785=1027.730,366.940,359.658,172.334,47.525,159.412
C00786=1027.738,367.186,359.618,172.341,47.526,159.413
C00787=1027.747,367.433,359.578,172.349,47.527,159.415
C00788=1027.755,367.680,359.538,172.356,47.528,159.416
C00789=1027.764,367.926,359.499,172.364,47.530,159.417
C00790=1027.772,368.173,359.460,172.372,47.531,159.419
C00791=1027.780,368.420,359.420,172.379,47.532,159.420
C00792=1027.788,368.666,359.380,172.387,47.534,159.421
C00793=1027.798,368.913,359.340,172.395,47.535,159.423
C00794=1027.805,369.160,359.300,172.402,47.536,159.424
C00795=1027.814,369.406,359.260,172.410,47.537,159.425
C00796=1027.822,369.653,359.220,172.419,47.538,159.427
C00797=1027.831,369.899,359.180,172.426,47.540,159.428
C00798=1027.839,370.147,359.140,172.434,47.541,159.429
C00799=1027.847,370.393,359.099,172.442,47.543,159.431
C00800=1027.856,370.639,359.059,172.449,47.544,159.432
C00801=1027.863,370.886,359.019,172.457,47.545,159.434
C00802=1027.872,371.133,358.978,172.465,47.547,159.435
C00803=1027.881,371.379,358.938,172.473,47.548,159.436
C00804=1027.888,371.626,358.898,172.480,47.550,159.438
C00805=1027.898,371.872,358.858,172.489,47.551,159.439
C00806=1027.906,372.119,358.817,172.497,47.553,159.441
C00807=1027.914,372.365,358.777,172.504,47.554,159.442
C00808=1027.923,372.612,358.737,172.512,47.556,159.444
C00809=1027.931,372.858,358.696,172.520,47.557,159.445
C00810=1027.940,373.105,358.656,172.528,47.559,159.446
C00811=1027.948,373.351,358.615,172.537,47.560,159.448
C00812=1027.957,373.598,358.574,172.545,47.562,159.449
C00813=1027.966,373.844,358.534,172.552,47.563,159.451
C00814=1027.974,374.091,358.493,172.560,47.565,159.452
C00815=1027.983,374.337,358.453,172.569,47.566,159.454
C00816=1027.992,374.584,358.412,172.577,47.568,159.455
C00817=1028.000,374.831,358.371,172.585,47.570,159.457
C00818=1028.009,375.077,358.331,172.592,47.571,159.458
C00819=1028.017,375.324,358.290,172.601,47.572,159.460
C00820=1028.026,375.571,358.249,172.609,47.574,159.461
C00821=1028.035,375.816,358.209,172.617,47.576,159.463
C00822=1028.044,376.063,358.168,172.626,47.577,159.464
C00823=1028.053,376.310,358.127,172.634,47.579,159.466
C00824=1028.061,376.556,358.087,172.642,47.581,159.467
C00825=1028.070,376.803,358.046,172.651,47.582,159.469
C00826=1028.079,377.049,358.004,172.659,47.584,159.470
C00827=1028.087,377.295,357.964,172.667,47.586,159.472
C00828=1028.096,377.542,357.923,172.676,47.587,159.473
C00829=1028.105,377.788,357.881,172.684,47.589,159.475
C00830=1028.113,378.035,357.840,172.692,47.591,159.477
C00831=1028.122,378.281,357.799,172.701,47.593,159.478
C00832=1028.131,378.528,357.757,172.709,47.595,159.480
C00833=1028.139,378.774,357.716,172.717,47.596,159.481
C00834=1028.148,379.020,357.675,172.726,47.598,159.483
C00835=1028.157,379.267,357.633,172.733,47.600,159.484
C00836=1028.165,379.499,357.595,172.741,47.602,159.486
C00837=1028.173,379.731,357.555,172.749,47.603,159.487
C00838=1028.182,379.963,357.516,172.757,47.605,159.489
C00839=1028.189,380.195,357.477,172.765,47.607,159.491
C00840=1028.198,380.428,357.438,172.774,47.609,159.492
C00841=1028.206,380.661,357.399,172.782,47.610,159.494
C00842=1028.214,380.892,357.360,172.790,47.612,159.495
C00843=1028.223,381.125,357.320,172.798,47.614,159.497
C00844=1028.232,381.371,357.278,172.806,47.616,159.498
C00845=1028.241,381.618,357.237,172.816,47.618,159.500
C00846=1028.249,381.864,357.195,172.823,47.620,159.502
C00847=1028.258,382.110,357.153,172.833,47.622,159.503
C00848=1028.267,382.357,357.112,172.842,47.624,159.505
C00849=1028.276,382.603,357.070,172.850,47.626,159.507
C00850=1028.285,382.849,357.028,172.859,47.627,159.508
C00851=1028.294,383.096,356.986,172.867,47.630,159.510
C00852=1028.303,383.342,356.944,172.877,47.632,159.512
C00853=1028.313,383.588,356.903,172.885,47.634,159.513
C00854=1028.322,383.834,356.861,172.894,47.636,159.515
C00855=1028.331,384.080,356.819,172.903,47.638,159.517
C00856=1028.340,384.326,356.777,172.911,47.640,159.519
C00857=1028.349,384.572,356.735,172.920,47.642,159.520
C00858=1028.358,384.819,356.694,172.930,47.644,159.522
C00859=1028.367,385.065,356.651,172.938,47.646,159.524
C00860=1028.377,385.312,356.609,172.947,47.649,159.526
C00861=1028.386,385.558,356.567,172.957,47.651,159.527
C00862=1028.395,385.804,356.525,172.965,47.653,159.529
C00863=1028.404,386.050,356.483,172.974,47.655,159.531
C00864=1028.413,386.296,356.441,172.983,47.657,159.533
C00865=1028.423,386.542,356.398,172.993,47.659,159.534
C00866=1028.431,386.789,356.356,173.001,47.662,159.536
C00867=1028.440,387.035,356.313,173.010,47.664,159.538
C00868=1028.450,387.281,356.270,173.020,47.666,159.540
C00869=1028.459,387.527,356.228,173.029,47.668,159.542
C00870=1028.468,387.774,356.186,173.037,47.670,159.543
C00871=1028.477,388.019,356.143,173.047,47.672,159.545
C00872=1028.487,388.266,356.100,173.056,47.675,159.547
C00873=1028.496,388.511,356.058,173.066,47.677,159.549
C00874=1028.504,388.758,356.015,173.075,47.679,159.551
C00875=1028.514,389.004,355.972,173.084,47.682,159.553
C00876=1028.524,389.250,355.930,173.093,47.684,159.555
C00877=1028.533,389.496,355.887,173.102,47.686,159.556
C00878=1028.542,389.742,355.844,173.112,47.689,159.558
C00879=1028.552,389.989,355.801,173.121,47.691,159.560
C00880=1028.561,390.234,355.759,173.131,47.694,159.562
C00881=1028.570,390.480,355.715,173.140,47.696,159.564
C00882=1028.580,390.726,355.672,173.149,47.699,159.566
C00883=1028.589,390.973,355.629,173.158,47.701,159.568
C00884=1028.598,391.218,355.586,173.168,47.704,159.570
C00885=1028.608,391.465,355.543,173.177,47.706,159.572
C00886=1028.617,391.711,355.500,173.187,47.709,159.574
C00887=1028.627,391.957,355.456,173.197,47.711,159.576
C00888=1028.635,392.203,355.413,173.206,47.714,159.578
C00889=1028.645,392.448,355.370,173.215,47.716,159.580
C00890=1028.655,392.695,355.326,173.225,47.719,159.582
C00891=1028.664,392.940,355.283,173.235,47.721,159.584
C00892=1028.674,393.187,355.240,173.244,47.724,159.586
C00893=1028.683,393.433,355.196,173.254,47.727,159.588
C00894=1028.693,393.678,355.153,173.264,47.729,159.590
C00895=1028.702,393.925,355.110,173.273,47.732,159.592
C00896=1028.712,394.179,355.064,173.284,47.734,159.594
C00897=1028.722,394.433,355.019,173.294,47.738,159.596
C00898=1028.732,394.688,354.974,173.304,47.740,159.598
C00899=1028.742,394.943,354.928,173.315,47.743,159.600
C00900=1028.751,395.188,354.885,173.324,47.746,159.602
C00901=1028.761,395.434,354.841,173.334,47.748,159.604
C00902=1028.771,395.680,354.798,173.344,47.751,159.606
C00903=1028.780,395.926,354.754,173.354,47.754,159.608
C00904=1028.790,396.172,354.709,173.364,47.756,159.610
C00905=1028.800,396.418,354.666,173.374,47.759,159.612
C00906=1028.809,396.664,354.622,173.384,47.762,159.615
C00907=1028.819,396.909,354.579,173.393,47.765,159.617
C00908=1028.828,397.155,354.534,173.403,47.768,159.619
C00909=1028.838,397.401,354.490,173.414,47.770,159.621
C00910=1028.848,397.647,354.446,173.424,47.774,159.623
C00911=1028.858,397.892,354.401,173.434,47.776,159.625
C00912=1028.868,398.138,354.358,173.444,47.779,159.627
C00913=1028.877,398.384,354.314,173.455,47.782,159.630
C00914=1028.887,398.630,354.269,173.464,47.785,159.632
C00915=1028.898,398.876,354.225,173.474,47.788,159.634
C00916=1028.907,399.122,354.180,173.485,47.791,159.636
C00917=1028.917,399.368,354.136,173.495,47.794,159.638
C00918=1028.927,399.614,354.091,173.505,47.797,159.640
C00919=1028.937,399.859,354.047,173.516,47.800,159.643
C00920=1028.946,400.105,354.003,173.526,47.803,159.645
C00921=1028.956,400.350,353.958,173.537,47.806,159.647
C00922=1028.966,400.596,353.913,173.547,47.809,159.649
C00923=1028.976,400.842,353.868,173.558,47.812,159.652
C00924=1028.986,401.088,353.823,173.568,47.815,159.654
C00925=1028.996,401.333,353.780,173.578,47.818,159.656
C00926=1029.006,401.579,353.735,173.589,47.821,159.658
C00927=1029.016,401.825,353.690,173.599,47.824,159.661
C00928=1029.026,402.071,353.645,173.610,47.827,159.663
C00929=1029.036,402.316,353.600,173.621,47.831,159.665
C00930=1029.046,402.562,353.554,173.632,47.834,159.668
C00931=1029.056,402.807,353.509,173.642,47.838,159.670
C00932=1029.066,403.053,353.465,173.653,47.840,159.672
C00933=1029.076,403.299,353.419,173.664,47.843,159.675
C00934=1029.086,403.545,353.375,173.674,47.847,159.677
C00935=1029.096,403.790,353.329,173.685,47.850,159.679
C00936=1029.106,404.036,353.284,173.696,47.853,159.682
C00937=1029.117,404.281,353.238,173.707,47.857,159.684
C00938=1029.126,404.527,353.193,173.718,47.860,159.686
C00939=1029.137,404.773,353.148,173.728,47.863,159.689
C00940=1029.147,405.018,353.102,173.740,47.867,159.691
C00941=1029.157,405.264,353.057,173.751,47.870,159.694
C00942=1029.167,405.509,353.012,173.761,47.873,159.696
C00943=1029.178,405.755,352.966,173.772,47.877,159.699
C00944=1029.188,406.001,352.921,173.784,47.880,159.701
C00945=1029.198,406.246,352.875,173.795,47.883,159.703
C00946=1029.208,406.492,352.829,173.805,47.887,159.706
C00947=1029.218,406.738,352.783,173.817,47.890,159.708
C00948=1029.229,406.983,352.737,173.828,47.894,159.711
C00949=1029.239,407.228,352.692,173.839,47.897,159.713
C00950=1029.249,407.474,352.646,173.851,47.901,159.716
C00951=1029.260,407.719,352.600,173.862,47.904,159.718
C00952=1029.271,407.965,352.554,173.872,47.908,159.721
C00953=1029.281,408.211,352.508,173.884,47.911,159.723
C00954=1029.292,408.456,352.462,173.895,47.915,159.726
C00955=1029.302,408.701,352.417,173.907,47.918,159.728
C00956=1029.314,408.971,352.367,173.919,47.922,159.731
C00957=1029.325,409.240,352.316,173.932,47.926,159.734
C00958=1029.342,409.628,352.243,173.950,47.932,159.738
C00959=1029.359,410.014,352.170,173.968,47.937,159.742
C00960=1029.376,410.401,352.098,173.987,47.943,159.746
C00961=1029.392,410.788,352.024,174.005,47.949,159.750
C00962=1029.403,411.033,351.978,174.016,47.953,159.753
C00963=1029.414,411.279,351.931,174.029,47.956,159.756
C00964=1029.424,411.524,351.884,174.041,47.960,159.759
C00965=1029.435,411.769,351.838,174.052,47.964,159.761
C00966=1029.446,412.015,351.792,174.064,47.968,159.764
C00967=1029.456,412.260,351.744,174.076,47.972,159.767
C00968=1029.467,412.505,351.698,174.087,47.976,159.769
C00969=1029.477,412.751,351.650,174.099,47.980,159.772
C00970=1029.488,412.997,351.604,174.112,47.983,159.775
C00971=1029.499,413.242,351.558,174.123,47.987,159.777
C00972=1029.510,413.488,351.510,174.135,47.991,159.780
C00973=1029.521,413.733,351.464,174.148,47.995,159.783
C00974=1029.532,413.978,351.417,174.160,47.999,159.786
C00975=1029.542,414.224,351.369,174.172,48.003,159.789
C00976=1029.554,414.468,351.322,174.184,48.006,159.791
C00977=1029.564,414.713,351.275,174.196,48.011,159.794
C00978=1029.575,414.959,351.228,174.208,48.015,159.797
C00979=1029.586,415.204,351.181,174.221,48.019,159.800
C00980=1029.597,415.450,351.134,174.233,48.023,159.803
C00981=1029.608,415.694,351.086,174.246,48.027,159.806
C00982=1029.619,415.940,351.039,174.258,48.031,159.808
C00983=1029.631,416.186,350.992,174.271,48.035,159.811
C00984=1029.643,416.431,350.944,174.283,48.039,159.814
C00985=1029.653,416.676,350.897,174.296,48.043,159.817
C00986=1029.664,416.922,350.848,174.308,48.047,159.820
C00987=1029.675,417.166,350.801,174.321,48.052,159.823
C00988=1029.686,417.412,350.754,174.333,48.056,159.826
C00989=1029.697,417.657,350.705,174.346,48.060,159.829
C00990=1029.708,417.902,350.658,174.358,48.064,159.832
C00991=1029.719,418.147,350.610,174.371,48.068,159.835
C00992=1029.730,418.392,350.561,174.384,48.073,159.838
C00993=1029.742,418.638,350.514,174.396,48.077,159.841
C00994=1029.753,418.882,350.466,174.409,48.081,159.844
C00995=1029.764,419.128,350.417,174.423,48.086,159.847
C00996=1029.776,419.373,350.370,174.436,48.090,159.850
C00997=1029.787,419.618,350.321,174.448,48.094,159.853
C00998=1029.798,419.863,350.273,174.461,48.099,159.856
C00999=1029.810,420.108,350.225,174.474,48.103,159.859
C01000=1029.821,420.353,350.176,174.488,48.107,159.862
C01001=1029.832,420.599,350.128,174.501,48.112,159.865
C01002=1029.844,420.844,350.080,174.514,48.116,159.868
C01003=1029.855,421.088,350.031,174.527,48.121,159.871
C01004=1029.867,421.334,349.983,174.540,48.125,159.875
C01005=1029.878,421.579,349.935,174.553,48.129,159.878
C01006=1029.890,421.823,349.886,174.567,48.134,159.881
C01007=1029.901,422.068,349.837,174.580,48.138,159.884
C01008=1029.914,422.314,349.789,174.593,48.143,159.887
C01009=1029.925,422.559,349.740,174.607,48.147,159.890
C01010=1029.936,422.803,349.691,174.621,48.152,159.894
C01011=1029.948,423.049,349.643,174.635,48.156,159.897
C01012=1029.960,423.293,349.595,174.648,48.161,159.900
C01013=1029.972,423.539,349.545,174.662,48.166,159.903
C01014=1029.985,423.825,349.487,174.678,48.171,159.907
C01015=1029.999,424.111,349.430,174.693,48.177,159.911
C01016=1030.012,424.398,349.372,174.710,48.182,159.915
C01017=1030.026,424.684,349.316,174.726,48.187,159.919
C01018=1030.038,424.929,349.266,174.740,48.193,159.922
C01019=1030.050,425.174,349.217,174.754,48.198,159.925
C01020=1030.062,425.419,349.167,174.768,48.202,159.929
C01021=1030.073,425.663,349.118,174.782,48.207,159.932
C01022=1030.085,425.909,349.068,174.796,48.212,159.935
C01023=1030.097,426.154,349.019,174.810,48.217,159.939
C01024=1030.109,426.398,348.969,174.824,48.221,159.942
C01025=1030.122,426.644,348.920,174.839,48.226,159.946
C01026=1030.134,426.888,348.871,174.852,48.231,159.949
C01027=1030.145,427.133,348.820,174.867,48.236,159.953
C01028=1030.157,427.377,348.770,174.881,48.241,159.956
C01029=1030.169,427.622,348.721,174.896,48.246,159.960
C01030=1030.181,427.867,348.671,174.910,48.251,159.963
C01031=1030.194,428.112,348.621,174.925,48.256,159.967
C01032=1030.205,428.356,348.571,174.939,48.261,159.970
C01033=1030.218,428.601,348.521,174.954,48.266,159.974
C01034=1030.229,428.846,348.470,174.969,48.271,159.977
C01035=1030.241,429.091,348.420,174.983,48.276,159.981
C01036=1030.253,429.334,348.369,174.998,48.281,159.984
C01037=1030.266,429.579,348.319,175.013,48.287,159.988
C01038=1030.278,429.824,348.269,175.028,48.291,159.992
C01039=1030.290,430.069,348.219,175.042,48.297,159.995
C01040=1030.303,430.313,348.168,175.057,48.302,159.999
C01041=1030.315,430.558,348.118,175.072,48.307,160.003
C01042=1030.328,430.802,348.067,175.087,48.312,160.006
C01043=1030.340,431.047,348.017,175.103,48.317,160.010
C01044=1030.352,431.291,347.966,175.118,48.323,160.014
C01045=1030.365,431.536,347.915,175.133,48.328,160.017
C01046=1030.378,431.781,347.865,175.148,48.333,160.021
C01047=1030.390,432.025,347.814,175.163,48.338,160.025
C01048=1030.403,432.270,347.763,175.179,48.344,160.029
C01049=1030.416,432.514,347.712,175.194,48.349,160.032
C01050=1030.429,432.759,347.661,175.209,48.354,160.036
C01051=1030.441,433.003,347.611,175.225,48.360,160.040
C01052=1030.453,433.248,347.560,175.241,48.365,160.044
C01053=1030.467,433.492,347.508,175.256,48.370,160.048
C01054=1030.479,433.736,347.457,175.272,48.376,160.052
C01055=1030.492,433.981,347.406,175.287,48.382,160.056
C01056=1030.504,434.226,347.354,175.304,48.387,160.059
C01057=1030.517,434.469,347.303,175.319,48.392,160.063
C01058=1030.530,434.714,347.252,175.335,48.398,160.067
C01059=1030.543,434.959,347.201,175.351,48.403,160.071
C01060=1030.556,435.203,347.148,175.367,48.409,160.075
C01061=1030.569,435.447,347.097,175.383,48.415,160.079
C01062=1030.582,435.692,347.046,175.399,48.420,160.083
C01063=1030.595,435.936,346.993,175.415,48.426,160.087
C01064=1030.608,436.180,346.942,175.432,48.432,160.091
C01065=1030.620,436.425,346.890,175.448,48.437,160.095
C01066=1030.633,436.669,346.838,175.464,48.443,160.099
C01067=1030.647,436.913,346.786,175.481,48.448,160.103
C01068=1030.659,437.157,346.734,175.496,48.455,160.108
C01069=1030.673,437.402,346.682,175.513,48.460,160.111
C01070=1030.685,437.645,346.629,175.530,48.466,160.116
C01071=1030.699,437.889,346.577,175.547,48.471,160.120
C01072=1030.712,438.134,346.525,175.563,48.478,160.124
C01073=1030.725,438.378,346.473,175.580,48.483,160.128
C01074=1030.740,438.643,346.416,175.598,48.490,160.133
C01075=1030.754,438.908,346.359,175.617,48.496,160.137
C01076=1030.769,439.173,346.302,175.635,48.502,160.142
C01077=1030.784,439.438,346.245,175.654,48.509,160.147
C01078=1030.797,439.682,346.192,175.671,48.515,160.151
C01079=1030.810,439.927,346.139,175.688,48.521,160.155
C01080=1030.823,440.170,346.087,175.705,48.527,160.160
C01081=1030.837,440.414,346.033,175.722,48.533,160.164
C01082=1030.850,440.658,345.981,175.739,48.539,160.168
C01083=1030.864,440.903,345.927,175.756,48.545,160.173
C01084=1030.878,441.146,345.875,175.774,48.551,160.177
C01085=1030.891,441.390,345.821,175.792,48.557,160.182
C01086=1030.905,441.634,345.769,175.809,48.563,160.186
C01087=1030.919,441.878,345.715,175.827,48.570,160.190
C01088=1030.933,442.122,345.662,175.845,48.575,160.195
C01089=1030.946,442.365,345.609,175.862,48.582,160.199
C01090=1030.960,442.610,345.556,175.879,48.588,160.204
C01091=1030.974,442.853,345.502,175.898,48.594,160.209
C01092=1030.987,443.097,345.449,175.915,48.600,160.213
C01093=1031.002,443.341,345.396,175.934,48.606,160.217
C01094=1031.016,443.583,345.343,175.952,48.613,160.222
C01095=1031.031,443.826,345.290,175.970,48.619,160.227
C01096=1031.047,444.069,345.238,175.988,48.625,160.231
C01097=1031.062,444.313,345.186,176.007,48.631,160.236
C01098=1031.079,444.556,345.135,176.025,48.637,160.240
C01099=1031.095,444.801,345.085,176.043,48.643,160.245
C01100=1031.113,445.044,345.034,176.062,48.648,160.249
C01101=1031.131,445.289,344.983,176.081,48.654,160.254
C01102=1031.149,445.532,344.934,176.100,48.659,160.258
C01103=1031.168,445.776,344.885,176.118,48.664,160.263
C01104=1031.187,446.020,344.836,176.137,48.670,160.267
C01105=1031.207,446.265,344.788,176.156,48.675,160.272
C01106=1031.228,446.509,344.740,176.176,48.680,160.276
C01107=1031.248,446.753,344.692,176.195,48.685,160.280
C01108=1031.270,446.997,344.646,176.214,48.690,160.285
C01109=1031.292,447.242,344.598,176.233,48.696,160.290
C01110=1031.314,447.486,344.552,176.252,48.701,160.294
C01111=1031.337,447.732,344.506,176.272,48.706,160.298
C01112=1031.360,447.976,344.461,176.291,48.710,160.303
C01113=1031.383,448.221,344.416,176.311,48.715,160.307
C01114=1031.408,448.466,344.371,176.331,48.720,160.312
C01115=1031.433,448.710,344.326,176.351,48.724,160.316
C01116=1031.458,448.956,344.283,176.371,48.728,160.320
C01117=1031.484,449.200,344.240,176.391,48.733,160.325
C01118=1031.510,449.445,344.197,176.411,48.738,160.329
C01119=1031.538,449.691,344.154,176.431,48.742,160.334
C01120=1031.564,449.936,344.111,176.451,48.746,160.338
C01121=1031.592,450.181,344.071,176.472,48.750,160.342
C01122=1031.620,450.426,344.028,176.492,48.754,160.347
C01123=1031.649,450.672,343.988,176.512,48.758,160.351
C01124=1031.678,450.917,343.947,176.533,48.762,160.355
C01125=1031.708,451.162,343.907,176.554,48.766,160.360
C01126=1031.739,451.409,343.868,176.575,48.770,160.364
C01127=1031.769,451.653,343.828,176.595,48.774,160.368
C01128=1031.800,451.900,343.789,176.616,48.777,160.373
C01129=1031.831,452.145,343.751,176.638,48.781,160.377
C01130=1031.864,452.391,343.713,176.658,48.785,160.381
C01131=1031.897,452.636,343.675,176.680,48.788,160.386
C01132=1031.930,452.882,343.639,176.701,48.792,160.390
C01133=1031.964,453.128,343.601,176.722,48.795,160.394
C01134=1032.008,453.448,343.554,176.751,48.799,160.400
C01135=1031.727,453.514,343.223,176.754,48.864,160.421
C01136=1031.688,453.239,343.263,176.729,48.860,160.416
C01137=1031.654,452.994,343.299,176.708,48.857,160.411
C01138=1031.621,452.749,343.336,176.687,48.853,160.407
C01139=1031.587,452.503,343.374,176.665,48.850,160.403
C01140=1031.556,452.256,343.412,176.644,48.847,160.399
C01141=1031.523,452.012,343.450,176.623,48.843,160.394
C01142=1031.492,451.766,343.488,176.602,48.839,160.390
C01143=1031.461,451.520,343.527,176.581,48.836,160.386
C01144=1031.431,451.274,343.567,176.560,48.832,160.381
C01145=1031.401,451.029,343.607,176.539,48.829,160.377
C01146=1031.371,450.784,343.647,176.518,48.825,160.372
C01147=1031.342,450.538,343.688,176.497,48.821,160.368
C01148=1031.314,450.292,343.729,176.478,48.816,160.364
C01149=1031.286,450.048,343.770,176.457,48.813,160.360
C01150=1031.258,449.803,343.813,176.436,48.809,160.355
C01151=1031.231,449.557,343.855,176.416,48.805,160.351
C01152=1031.205,449.312,343.897,176.396,48.800,160.346
C01153=1031.179,449.067,343.941,176.376,48.796,160.342
C01154=1031.153,448.822,343.985,176.355,48.792,160.337
C01155=1031.128,448.577,344.028,176.335,48.787,160.333
C01156=1031.104,448.333,344.073,176.317,48.783,160.329
C01157=1031.079,448.087,344.118,176.297,48.778,160.324
C01158=1031.056,447.843,344.163,176.276,48.773,160.320
C01159=1031.033,447.598,344.208,176.258,48.769,160.315
C01160=1031.010,447.353,344.254,176.238,48.764,160.311
C01161=1030.988,447.109,344.301,176.218,48.759,160.307
C01162=1030.967,446.865,344.348,176.199,48.754,160.302
C01163=1030.945,446.620,344.395,176.179,48.749,160.298
C01164=1030.924,446.376,344.443,176.160,48.744,160.293
C01165=1030.904,446.132,344.490,176.141,48.739,160.289
C01166=1030.885,445.887,344.540,176.123,48.733,160.284
C01167=1030.866,445.643,344.589,176.104,48.728,160.280
C01168=1030.846,445.400,344.638,176.084,48.723,160.275
C01169=1030.829,445.155,344.688,176.066,48.717,160.271
C01170=1030.811,444.912,344.737,176.047,48.712,160.266
C01171=1030.794,444.668,344.789,176.029,48.706,160.262
C01172=1030.777,444.425,344.839,176.010,48.700,160.257
C01173=1030.761,444.180,344.891,175.992,48.695,160.253
C01174=1030.745,443.937,344.942,175.974,48.689,160.248
C01175=1030.730,443.694,344.995,175.955,48.683,160.244
C01176=1030.715,443.450,345.047,175.937,48.677,160.239
C01177=1030.701,443.207,345.101,175.920,48.671,160.235
C01178=1030.687,442.964,345.154,175.901,48.665,160.230
C01179=1030.673,442.721,345.206,175.884,48.659,160.226
C01180=1030.659,442.477,345.261,175.865,48.653,160.221
C01181=1030.645,442.233,345.313,175.848,48.646,160.217
C01182=1030.632,441.990,345.367,175.830,48.641,160.212
C01183=1030.617,441.745,345.420,175.812,48.634,160.208
C01184=1030.604,441.501,345.473,175.794,48.629,160.203
C01185=1030.591,441.258,345.526,175.777,48.622,160.199
C01186=1030.577,441.013,345.580,175.759,48.616,160.194
C01187=1030.563,440.769,345.632,175.741,48.611,160.190
C01188=1030.550,440.525,345.685,175.724,48.605,160.186
C01189=1030.536,440.282,345.738,175.707,48.599,160.181
C01190=1030.523,440.038,345.791,175.690,48.593,160.177
C01191=1030.509,439.794,345.844,175.673,48.587,160.173
C01192=1030.496,439.549,345.897,175.655,48.581,160.168
C01193=1030.481,439.283,345.954,175.637,48.575,160.164
C01194=1030.467,439.018,346.011,175.619,48.568,160.159
C01195=1030.452,438.751,346.069,175.600,48.562,160.154
C01196=1030.438,438.485,346.126,175.582,48.556,160.150
C01197=1030.424,438.242,346.178,175.565,48.550,160.146
C01198=1030.412,437.997,346.230,175.548,48.544,160.142
C01199=1030.398,437.753,346.282,175.531,48.538,160.137
C01200=1030.385,437.508,346.335,175.514,48.533,160.133
C01201=1030.371,437.265,346.387,175.498,48.527,160.129
C01202=1030.358,437.021,346.439,175.481,48.521,160.125
C01203=1030.346,436.777,346.491,175.465,48.516,160.121
C01204=1030.332,436.532,346.543,175.449,48.510,160.117
C01205=1030.320,436.287,346.595,175.432,48.504,160.113
C01206=1030.307,436.044,346.646,175.416,48.499,160.109
C01207=1030.293,435.799,346.698,175.400,48.493,160.105
C01208=1030.280,435.555,346.751,175.383,48.488,160.101
C01209=1030.268,435.310,346.802,175.368,48.482,160.097
C01210=1030.254,435.066,346.854,175.351,48.477,160.093
C01211=1030.242,434.822,346.905,175.336,48.471,160.089
C01212=1030.229,434.577,346.957,175.319,48.466,160.085
C01213=1030.216,434.333,347.008,175.303,48.460,160.081
C01214=1030.203,434.089,347.060,175.288,48.455,160.077
C01215=1030.191,433.844,347.111,175.272,48.450,160.073
C01216=1030.178,433.600,347.162,175.256,48.444,160.069
C01217=1030.165,433.355,347.213,175.241,48.439,160.065
C01218=1030.152,433.111,347.264,175.224,48.434,160.062
C01219=1030.139,432.866,347.315,175.209,48.429,160.058
C01220=1030.127,432.622,347.366,175.194,48.423,160.054
C01221=1030.115,432.377,347.417,175.178,48.418,160.050
C01222=1030.102,432.133,347.468,175.163,48.413,160.046
C01223=1030.089,431.888,347.519,175.148,48.407,160.043
C01224=1030.077,431.644,347.569,175.133,48.402,160.039
C01225=1030.064,431.399,347.620,175.117,48.397,160.035
C01226=1030.051,431.155,347.671,175.101,48.392,160.032
C01227=1030.039,430.910,347.721,175.086,48.387,160.028
C01228=1030.026,430.666,347.772,175.072,48.382,160.024
C01229=1030.014,430.421,347.822,175.057,48.376,160.020
C01230=1030.001,430.177,347.873,175.042,48.371,160.017
C01231=1029.990,429.932,347.923,175.027,48.367,160.013
C01232=1029.978,429.687,347.973,175.012,48.361,160.010
C01233=1029.965,429.442,348.024,174.996,48.356,160.006
C01234=1029.953,429.198,348.074,174.982,48.352,160.002
C01235=1029.940,428.953,348.124,174.967,48.346,159.999
C01236=1029.928,428.709,348.175,174.953,48.341,159.995
C01237=1029.916,428.464,348.224,174.938,48.337,159.992
C01238=1029.904,428.220,348.274,174.924,48.331,159.988
C01239=1029.892,427.975,348.324,174.909,48.326,159.985
C01240=1029.880,427.730,348.375,174.894,48.322,159.981
C01241=1029.868,427.485,348.425,174.880,48.317,159.978
C01242=1029.856,427.241,348.475,174.865,48.312,159.974
C01243=1029.845,426.996,348.524,174.852,48.307,159.971
C01244=1029.832,426.751,348.574,174.837,48.302,159.967
C01245=1029.820,426.506,348.624,174.823,48.297,159.964
C01246=1029.809,426.262,348.673,174.808,48.293,159.960
C01247=1029.796,426.017,348.723,174.794,48.288,159.957
C01248=1029.784,425.771,348.773,174.779,48.283,159.953
C01249=1029.773,425.527,348.822,174.766,48.278,159.950
C01250=1029.761,425.282,348.872,174.751,48.274,159.947
C01251=1029.748,425.037,348.920,174.738,48.269,159.944
C01252=1029.736,424.792,348.970,174.724,48.264,159.940
C01253=1029.723,424.503,349.028,174.707,48.259,159.936
C01254=1029.709,424.214,349.085,174.691,48.254,159.932
C01255=1029.695,423.926,349.144,174.675,48.248,159.928
C01256=1029.681,423.637,349.201,174.658,48.242,159.924
C01257=1029.670,423.392,349.250,174.645,48.238,159.921
C01258=1029.659,423.147,349.299,174.631,48.233,159.918
C01259=1029.646,422.902,349.348,174.617,48.229,159.915
C01260=1029.635,422.657,349.397,174.604,48.225,159.912
C01261=1029.623,422.412,349.446,174.590,48.220,159.908
C01262=1029.612,422.167,349.495,174.577,48.215,159.905
C01263=1029.599,421.922,349.543,174.563,48.211,159.902
C01264=1029.588,421.677,349.592,174.550,48.207,159.899
C01265=1029.577,421.432,349.641,174.537,48.202,159.896
C01266=1029.565,421.187,349.688,174.523,48.198,159.893
C01267=1029.554,420.942,349.737,174.510,48.194,159.890
C01268=1029.542,420.697,349.786,174.497,48.189,159.886
C01269=1029.531,420.452,349.833,174.483,48.185,159.883
C01270=1029.519,420.207,349.882,174.470,48.181,159.880
C01271=1029.508,419.962,349.931,174.457,48.177,159.877
C01272=1029.496,419.717,349.978,174.445,48.172,159.874
C01273=1029.485,419.471,350.027,174.432,48.168,159.871
C01274=1029.474,419.226,350.075,174.419,48.164,159.868
C01275=1029.462,418.981,350.123,174.405,48.159,159.865
C01276=1029.451,418.736,350.171,174.392,48.155,159.862
C01277=1029.441,418.491,350.219,174.380,48.151,159.859
C01278=1029.429,418.246,350.267,174.367,48.147,159.856
C01279=1029.418,418.001,350.315,174.354,48.143,159.853
C01280=1029.407,417.755,350.363,174.342,48.138,159.850
C01281=1029.396,417.510,350.410,174.329,48.134,159.847
C01282=1029.385,417.265,350.458,174.315,48.130,159.844
C01283=1029.373,417.020,350.506,174.303,48.126,159.841
C01284=1029.362,416.775,350.554,174.290,48.122,159.838
C01285=1029.351,416.529,350.601,174.278,48.118,159.835
C01286=1029.340,416.285,350.649,174.266,48.114,159.832
C01287=1029.329,416.039,350.696,174.252,48.110,159.829
C01288=1029.318,415.793,350.743,174.241,48.106,159.827
C01289=1029.307,415.548,350.791,174.228,48.102,159.824
C01290=1029.296,415.303,350.838,174.216,48.098,159.821
C01291=1029.285,415.058,350.885,174.203,48.094,159.818
C01292=1029.274,414.812,350.932,174.191,48.090,159.815
C01293=1029.263,414.567,350.980,174.178,48.087,159.813
C01294=1029.251,414.322,351.027,174.166,48.082,159.810
C01295=1029.241,414.076,351.074,174.155,48.078,159.807
C01296=1029.230,413.831,351.121,174.142,48.075,159.804
C01297=1029.219,413.586,351.168,174.130,48.071,159.801
C01298=1029.209,413.341,351.215,174.118,48.067,159.799
C01299=1029.197,413.095,351.262,174.105,48.063,159.796
C01300=1029.187,412.850,351.309,174.094,48.059,159.793
C01301=1029.176,412.605,351.356,174.082,48.055,159.790
C01302=1029.165,412.359,351.401,174.070,48.052,159.788
C01303=1029.154,412.113,351.449,174.058,48.048,159.785
C01304=1029.144,411.868,351.496,174.046,48.045,159.782
C01305=1029.133,411.623,351.542,174.034,48.041,159.780
C01306=1029.123,411.377,351.589,174.023,48.037,159.777
C01307=1029.112,411.132,351.635,174.010,48.033,159.774
C01308=1029.102,410.886,351.682,173.999,48.030,159.772
C01309=1029.091,410.641,351.729,173.987,48.026,159.769
C01310=1029.080,410.396,351.774,173.975,48.022,159.766
C01311=1029.070,410.150,351.822,173.964,48.019,159.764
C01312=1029.059,409.904,351.868,173.952,48.015,159.761
C01313=1029.047,409.627,351.920,173.939,48.011,159.758
C01314=1029.035,409.348,351.972,173.926,48.007,159.755
C01315=1029.023,409.069,352.024,173.913,48.003,159.752
C01316=1029.011,408.792,352.077,173.900,48.000,159.750
C01317=1029.000,408.546,352.123,173.888,47.996,159.747
C01318=1028.990,408.301,352.168,173.877,47.992,159.744
C01319=1028.979,408.055,352.214,173.866,47.989,159.742
C01320=1028.969,407.809,352.260,173.855,47.985,159.739
C01321=1028.958,407.564,352.306,173.843,47.982,159.737
C01322=1028.947,407.318,352.352,173.832,47.979,159.734
C01323=1028.938,407.073,352.397,173.821,47.975,159.732
C01324=1028.927,406.827,352.443,173.809,47.972,159.729
C01325=1028.916,406.581,352.489,173.798,47.969,159.727
C01326=1028.906,406.336,352.535,173.787,47.965,159.724
C01327=1028.896,406.090,352.579,173.775,47.962,159.722
C01328=1028.885,405.845,352.625,173.765,47.958,159.720
C01329=1028.875,405.599,352.671,173.754,47.955,159.717
C01330=1028.865,405.354,352.716,173.743,47.952,159.715
C01331=1028.854,405.108,352.762,173.731,47.949,159.712
C01332=1028.845,404.863,352.807,173.721,47.946,159.710
C01333=1028.834,404.617,352.853,173.710,47.942,159.708
C01334=1028.824,404.371,352.898,173.698,47.939,159.705
C01335=1028.814,404.126,352.943,173.688,47.936,159.703
C01336=1028.804,403.880,352.988,173.677,47.932,159.700
C01337=1028.794,403.634,353.033,173.666,47.929,159.698
C01338=1028.784,403.389,353.079,173.656,47.926,159.696
C01339=1028.773,403.143,353.124,173.645,47.923,159.693
C01340=1028.764,402.898,353.169,173.634,47.920,159.691
C01341=1028.753,402.651,353.214,173.623,47.916,159.689
C01342=1028.743,402.406,353.260,173.612,47.914,159.686
C01343=1028.734,402.161,353.305,173.602,47.910,159.684
C01344=1028.724,401.915,353.349,173.591,47.908,159.682
C01345=1028.714,401.669,353.395,173.581,47.904,159.680
C01346=1028.704,401.424,353.439,173.570,47.902,159.677
C01347=1028.694,401.178,353.484,173.559,47.898,159.675
C01348=1028.684,400.931,353.529,173.549,47.895,159.673
C01349=1028.675,400.710,353.569,173.539,47.893,159.671
C01350=1028.666,400.488,353.610,173.530,47.890,159.669
C01351=1028.657,400.266,353.649,173.521,47.887,159.667
C01352=1028.649,400.044,353.690,173.511,47.885,159.665
C01353=1028.639,399.822,353.731,173.502,47.882,159.663
C01354=1028.630,399.599,353.771,173.493,47.879,159.661
C01355=1028.621,399.377,353.811,173.483,47.877,159.659
C01356=1028.612,399.155,353.850,173.474,47.874,159.657
C01357=1028.603,398.910,353.895,173.464,47.871,159.655
C01358=1028.593,398.664,353.939,173.453,47.869,159.652
C01359=1028.583,398.418,353.984,173.443,47.865,159.650
C01360=1028.573,398.172,354.028,173.433,47.863,159.648
C01361=1028.564,397.926,354.072,173.422,47.860,159.646
C01362=1028.553,397.681,354.116,173.413,47.857,159.644
C01363=1028.544,397.435,354.160,173.403,47.854,159.641
C01364=1028.535,397.189,354.204,173.392,47.852,159.639
C01365=1028.524,396.943,354.248,173.382,47.849,159.637
C01366=1028.515,396.698,354.293,173.372,47.846,159.635
C01367=1028.505,396.452,354.336,173.363,47.843,159.633
C01368=1028.495,396.206,354.380,173.352,47.841,159.631
C01369=1028.486,395.959,354.424,173.342,47.838,159.629
C01370=1028.476,395.714,354.468,173.332,47.835,159.627
C01371=1028.466,395.467,354.512,173.323,47.833,159.625
C01372=1028.457,395.222,354.555,173.312,47.830,159.623
C01373=1028.445,394.917,354.609,173.300,47.826,159.620
C01374=1028.433,394.614,354.663,173.288,47.823,159.618
C01375=1028.422,394.310,354.717,173.276,47.820,159.615
C01376=1028.409,394.005,354.772,173.264,47.817,159.613
C01377=1028.401,393.759,354.815,173.254,47.815,159.611
C01378=1028.391,393.514,354.858,173.244,47.812,159.609
C01379=1028.381,393.267,354.902,173.235,47.810,159.607
C01380=1028.371,393.021,354.945,173.225,47.807,159.605
C01381=1028.362,392.776,354.988,173.215,47.804,159.603
C01382=1028.353,392.529,355.032,173.206,47.802,159.601
C01383=1028.343,392.284,355.075,173.195,47.800,159.599
C01384=1028.334,392.037,355.118,173.186,47.797,159.597
C01385=1028.324,391.791,355.162,173.176,47.795,159.595
C01386=1028.315,391.546,355.204,173.167,47.793,159.593
C01387=1028.305,391.300,355.248,173.157,47.790,159.591
C01388=1028.296,391.054,355.291,173.147,47.787,159.589
C01389=1028.287,390.807,355.334,173.138,47.785,159.587
C01390=1028.277,390.562,355.377,173.128,47.783,159.585
C01391=1028.267,390.316,355.420,173.120,47.780,159.583
C01392=1028.259,390.069,355.463,173.110,47.778,159.581
C01393=1028.249,389.823,355.506,173.101,47.776,159.579
C01394=1028.241,389.577,355.549,173.091,47.773,159.577
C01395=1028.231,389.331,355.592,173.082,47.771,159.576
C01396=1028.222,389.085,355.634,173.073,47.769,159.574
C01397=1028.212,388.839,355.677,173.063,47.766,159.572
C01398=1028.203,388.592,355.720,173.054,47.764,159.570
C01399=1028.194,388.347,355.762,173.045,47.762,159.568
C01400=1028.185,388.101,355.805,173.036,47.760,159.566
C01401=1028.175,387.854,355.848,173.027,47.758,159.565
C01402=1028.166,387.608,355.891,173.018,47.755,159.563
C01403=1028.157,387.363,355.933,173.008,47.753,159.561
C01404=1028.147,387.116,355.976,172.999,47.751,159.559
C01405=1028.138,386.870,356.018,172.989,47.749,159.557
C01406=1028.130,386.624,356.061,172.981,47.746,159.555
C01407=1028.121,386.378,356.103,172.972,47.744,159.554
C01408=1028.111,386.131,356.145,172.962,47.742,159.552
C01409=1028.102,385.885,356.188,172.953,47.741,159.550
C01410=1028.093,385.639,356.229,172.945,47.738,159.549
C01411=1028.084,385.393,356.272,172.936,47.736,159.547
C01412=1028.074,385.146,356.314,172.926,47.734,159.545
C01413=1028.065,384.900,356.356,172.917,47.732,159.543
C01414=1028.056,384.654,356.398,172.909,47.730,159.542
C01415=1028.046,384.408,356.439,172.900,47.728,159.540
C01416=1028.037,384.161,356.481,172.890,47.726,159.538
C01417=1028.028,383.916,356.523,172.882,47.724,159.536
C01418=1028.019,383.669,356.565,172.873,47.722,159.535
C01419=1028.010,383.423,356.607,172.864,47.720,159.533
C01420=1028.001,383.177,356.648,172.856,47.718,159.531
C01421=1027.992,382.930,356.690,172.847,47.716,159.529
C01422=1027.983,382.684,356.733,172.838,47.715,159.528
C01423=1027.974,382.438,356.774,172.829,47.712,159.526
C01424=1027.965,382.192,356.816,172.820,47.711,159.524
C01425=1027.956,381.945,356.858,172.812,47.709,159.523
C01426=1027.947,381.699,356.899,172.803,47.707,159.521
C01427=1027.938,381.453,356.941,172.794,47.705,159.520
C01428=1027.930,381.206,356.983,172.786,47.703,159.518
C01429=1027.921,380.972,357.022,172.778,47.701,159.516
C01430=1027.913,380.739,357.061,172.769,47.699,159.515
C01431=1027.904,380.506,357.101,172.761,47.698,159.513
C01432=1027.896,380.273,357.140,172.753,47.696,159.512
C01433=1027.888,380.039,357.180,172.745,47.695,159.510
C01434=1027.880,379.806,357.219,172.737,47.693,159.509
C01435=1027.871,379.572,357.259,172.729,47.691,159.507
C01436=1027.863,379.339,357.297,172.721,47.689,159.506
C01437=1027.854,379.092,357.338,172.712,47.688,159.504
C01438=1027.845,378.846,357.380,172.704,47.686,159.502
C01439=1027.837,378.600,357.421,172.695,47.684,159.501
C01440=1027.828,378.353,357.462,172.687,47.682,159.499
C01441=1027.819,378.107,357.504,172.678,47.681,159.498
C01442=1027.810,377.861,357.546,172.670,47.679,159.496
C01443=1027.802,377.614,357.586,172.662,47.677,159.495
C01444=1027.793,377.368,357.628,172.653,47.676,159.493
C01445=1027.785,377.122,357.669,172.645,47.674,159.491
C01446=1027.777,376.875,357.710,172.636,47.672,159.490
C01447=1027.767,376.629,357.751,172.629,47.671,159.488
C01448=1027.758,376.382,357.792,172.621,47.669,159.487
C01449=1027.750,376.136,357.832,172.612,47.668,159.485
C01450=1027.741,375.889,357.873,172.604,47.666,159.484
C01451=1027.733,375.643,357.913,172.595,47.665,159.482
C01452=1027.723,375.396,357.955,172.587,47.663,159.481
C01453=1027.715,375.149,357.996,172.579,47.661,159.479
C01454=1027.707,374.903,358.036,172.571,47.660,159.478
C01455=1027.697,374.657,358.077,172.563,47.658,159.476
C01456=1027.689,374.410,358.117,172.555,47.657,159.475
C01457=1027.680,374.164,358.158,172.547,47.655,159.473
C01458=1027.672,373.917,358.198,172.538,47.654,159.472
C01459=1027.663,373.670,358.239,172.530,47.653,159.470
C01460=1027.654,373.424,358.279,172.523,47.651,159.469
C01461=1027.646,373.177,358.320,172.514,47.650,159.468
C01462=1027.637,372.931,358.360,172.506,47.648,159.466
C01463=1027.629,372.684,358.400,172.498,47.647,159.465
C01464=1027.621,372.437,358.441,172.490,47.645,159.463
C01465=1027.612,372.192,358.481,172.483,47.644,159.462
C01466=1027.604,371.945,358.522,172.474,47.643,159.461
C01467=1027.595,371.698,358.562,172.466,47.641,159.459
C01468=1027.587,371.452,358.602,172.459,47.640,159.458
C01469=1027.579,371.205,358.643,172.451,47.639,159.456
C01470=1027.570,370.958,358.683,172.443,47.637,159.455
C01471=1027.562,370.712,358.723,172.434,47.636,159.453
C01472=1027.553,370.466,358.763,172.427,47.635,159.452
C01473=1027.545,370.218,358.804,172.419,47.633,159.451
C01474=1027.537,369.972,358.844,172.411,47.632,159.449
C01475=1027.528,369.725,358.884,172.404,47.631,159.448
C01476=1027.520,369.479,358.924,172.396,47.630,159.447
C01477=1027.512,369.232,358.964,172.388,47.628,159.445
C01478=1027.503,368.985,359.005,172.381,47.627,159.444
C01479=1027.495,368.739,359.044,172.372,47.626,159.443
C01480=1027.487,368.492,359.084,172.364,47.625,159.441
C01481=1027.478,368.245,359.123,172.357,47.623,159.440
C01482=1027.470,367.999,359.163,172.349,47.622,159.438
C01483=1027.461,367.752,359.203,172.342,47.621,159.437
C01484=1027.453,367.505,359.243,172.334,47.620,159.436
C01485=1027.444,367.259,359.282,172.327,47.619,159.435
C01486=1027.436,367.012,359.321,172.319,47.618,159.433
C01487=1027.428,366.765,359.361,172.311,47.616,159.432
C01488=1027.420,366.518,359.401,172.304,47.616,159.431
C01489=1027.412,366.296,359.436,172.296,47.614,159.429
C01490=1027.405,366.074,359.473,172.290,47.614,159.428
C01491=1027.397,365.850,359.508,172.283,47.613,159.427
C01492=1027.389,365.628,359.544,172.276,47.612,159.426
C01493=1027.382,365.404,359.579,172.269,47.611,159.425
C01494=1027.375,365.182,359.615,172.262,47.610,159.424
C01495=1027.367,364.959,359.650,172.256,47.609,159.423
C01496=1027.360,364.736,359.686,172.249,47.608,159.421
C01497=1027.351,364.490,359.725,172.242,47.607,159.420
C01498=1027.344,364.243,359.765,172.234,47.606,159.419
C01499=1027.335,363.996,359.804,172.227,47.605,159.418
C01500=1027.327,363.750,359.844,172.219,47.604,159.416
C01501=1027.319,363.502,359.882,172.212,47.603,159.415
C01502=1027.311,363.255,359.922,172.204,47.602,159.414
C01503=1027.303,363.009,359.961,172.198,47.601,159.413
C01504=1027.295,362.762,360.000,172.190,47.600,159.412
C01505=1027.286,362.516,360.039,172.183,47.599,159.410
C01506=1027.279,362.269,360.079,172.175,47.598,159.409
C01507=1027.271,362.022,360.118,172.168,47.597,159.408
C01508=1027.262,361.775,360.157,172.160,47.596,159.407
C01509=1027.255,361.528,360.195,172.153,47.596,159.406
C01510=1027.247,361.282,360.235,172.145,47.594,159.404
C01511=1027.239,361.034,360.274,172.138,47.594,159.403
C01512=1027.230,360.788,360.313,172.132,47.593,159.402
C01513=1027.223,360.541,360.351,172.124,47.592,159.401
C01514=1027.214,360.295,360.391,172.117,47.591,159.400
C01515=1027.206,360.047,360.429,172.110,47.591,159.399
C01516=1027.198,359.800,360.468,172.103,47.590,159.397
C01517=1027.190,359.554,360.507,172.095,47.589,159.396
C01518=1027.182,359.307,360.545,172.088,47.588,159.395
C01519=1027.174,359.060,360.584,172.081,47.587,159.394
C01520=1027.166,358.813,360.623,172.074,47.586,159.393
C01521=1027.158,358.566,360.661,172.067,47.586,159.392
C01522=1027.150,358.319,360.699,172.060,47.586,159.391
C01523=1027.141,358.072,360.739,172.052,47.585,159.389
C01524=1027.134,357.826,360.777,172.046,47.584,159.388
C01525=1027.126,357.579,360.816,172.039,47.583,159.387
C01526=1027.118,357.332,360.854,172.031,47.582,159.386
C01527=1027.110,357.085,360.892,172.024,47.582,159.385
C01528=1027.102,356.838,360.931,172.017,47.581,159.384
C01529=1027.094,356.591,360.969,172.011,47.581,159.383
C01530=1027.086,356.344,361.008,172.003,47.580,159.382
C01531=1027.078,356.097,361.045,171.996,47.579,159.381
C01532=1027.070,355.850,361.083,171.989,47.578,159.379
C01533=1027.063,355.603,361.122,171.983,47.578,159.378
C01534=1027.054,355.356,361.160,171.975,47.577,159.377
C01535=1027.047,355.110,361.199,171.968,47.577,159.376
C01536=1027.039,354.862,361.237,171.962,47.576,159.375
C01537=1027.031,354.615,361.275,171.955,47.576,159.374
C01538=1027.023,354.368,361.313,171.948,47.575,159.373
C01539=1027.015,354.122,361.351,171.941,47.575,159.372
C01540=1027.007,353.874,361.389,171.934,47.574,159.371
C01541=1027.000,353.628,361.427,171.927,47.574,159.370
C01542=1026.991,353.380,361.464,171.920,47.573,159.369
C01543=1026.983,353.133,361.503,171.914,47.573,159.368
C01544=1026.975,352.886,361.541,171.907,47.572,159.367
C01545=1026.968,352.639,361.579,171.900,47.572,159.366
C01546=1026.960,352.393,361.616,171.894,47.571,159.365
C01547=1026.952,352.145,361.654,171.886,47.571,159.364
C01548=1026.945,351.898,361.692,171.879,47.571,159.363
C01549=1026.937,351.679,361.726,171.873,47.570,159.362
C01550=1026.931,351.459,361.759,171.867,47.570,159.361
C01551=1026.923,351.240,361.793,171.861,47.569,159.360
C01552=1026.916,351.020,361.826,171.855,47.569,159.359
C01553=1026.910,350.801,361.859,171.849,47.569,159.358
C01554=1026.903,350.581,361.894,171.843,47.568,159.357
C01555=1026.896,350.361,361.927,171.837,47.568,159.357
C01556=1026.889,350.142,361.960,171.831,47.567,159.356
C01557=1026.882,349.896,361.998,171.825,47.567,159.355
C01558=1026.873,349.648,362.035,171.818,47.567,159.354
C01559=1026.866,349.401,362.073,171.812,47.566,159.353
C01560=1026.859,349.154,362.110,171.805,47.566,159.352
C01561=1026.851,348.907,362.147,171.798,47.566,159.351
C01562=1026.843,348.659,362.185,171.792,47.565,159.350
C01563=1026.836,348.413,362.223,171.785,47.565,159.349
C01564=1026.828,348.166,362.260,171.779,47.565,159.348
C01565=1026.820,347.919,362.298,171.772,47.565,159.347
C01566=1026.812,347.672,362.335,171.766,47.564,159.346
C01567=1026.805,347.425,362.372,171.759,47.564,159.345
C01568=1026.796,347.177,362.410,171.752,47.564,159.344
C01569=1026.790,346.929,362.446,171.746,47.564,159.343
C01570=1026.782,346.683,362.483,171.739,47.563,159.342
C01571=1026.774,346.436,362.520,171.733,47.563,159.342
C01572=1026.766,346.189,362.558,171.726,47.563,159.341
C01573=1026.758,345.942,362.595,171.720,47.563,159.340
C01574=1026.751,345.695,362.632,171.714,47.563,159.339
C01575=1026.743,345.447,362.669,171.708,47.563,159.338
C01576=1026.736,345.200,362.706,171.701,47.562,159.337
C01577=1026.728,344.953,362.743,171.695,47.562,159.336
C01578=1026.721,344.706,362.781,171.688,47.562,159.335
C01579=1026.713,344.459,362.817,171.682,47.562,159.334
C01580=1026.705,344.212,362.854,171.675,47.562,159.334
C01581=1026.698,343.965,362.891,171.669,47.562,159.333
C01582=1026.690,343.717,362.927,171.662,47.562,159.332
C01583=1026.683,343.470,362.965,171.656,47.562,159.331
C01584=1026.675,343.223,363.001,171.650,47.561,159.330
C01585=1026.667,342.976,363.038,171.643,47.561,159.329
C01586=1026.660,342.729,363.076,171.638,47.561,159.328
C01587=1026.653,342.481,363.112,171.631,47.561,159.327
C01588=1026.645,342.235,363.149,171.625,47.561,159.327
C01589=1026.638,341.987,363.186,171.618,47.561,159.326
C01590=1026.630,341.739,363.222,171.612,47.561,159.325
C01591=1026.622,341.493,363.259,171.605,47.561,159.324
C01592=1026.615,341.245,363.296,171.599,47.561,159.323
C01593=1026.608,340.999,363.332,171.594,47.561,159.322
C01594=1026.600,340.751,363.368,171.587,47.561,159.322
C01595=1026.593,340.503,363.405,171.581,47.561,159.321
C01596=1026.585,340.257,363.442,171.574,47.561,159.320
C01597=1026.577,340.009,363.478,171.568,47.561,159.319
C01598=1026.570,339.762,363.514,171.563,47.562,159.318
C01599=1026.563,339.515,363.551,171.556,47.561,159.317
C01600=1026.556,339.267,363.587,171.550,47.562,159.317
C01601=1026.548,339.020,363.623,171.543,47.562,159.316
C01602=1026.540,338.773,363.660,171.537,47.562,159.315
C01603=1026.533,338.526,363.696,171.532,47.562,159.314
C01604=1026.525,338.279,363.732,171.525,47.562,159.314
C01605=1026.518,338.031,363.769,171.519,47.562,159.313
C01606=1026.510,337.784,363.805,171.513,47.562,159.312
C01607=1026.503,337.537,363.841,171.507,47.563,159.311
C01608=1026.495,337.290,363.877,171.501,47.563,159.311
C01609=1026.489,337.069,363.909,171.495,47.563,159.310
C01610=1026.483,336.848,363.942,171.490,47.563,159.309
C01611=1026.476,336.626,363.974,171.485,47.563,159.308
C01612=1026.469,336.405,364.006,171.479,47.563,159.308
C01613=1026.462,336.184,364.039,171.474,47.564,159.307
C01614=1026.456,335.963,364.070,171.468,47.564,159.306
C01615=1026.449,335.742,364.102,171.462,47.564,159.306
C01616=1026.443,335.521,364.135,171.458,47.564,159.305
C01617=1026.435,335.274,364.171,171.451,47.564,159.304
C01618=1026.428,335.026,364.206,171.445,47.565,159.304
C01619=1026.420,334.779,364.242,171.439,47.565,159.303
C01620=1026.413,334.531,364.279,171.434,47.565,159.302
C01621=1026.406,334.284,364.315,171.427,47.565,159.301
C01622=1026.399,334.036,364.351,171.421,47.566,159.301
C01623=1026.392,333.789,364.387,171.416,47.566,159.300
C01624=1026.384,333.542,364.423,171.409,47.566,159.299
C01625=1026.378,333.295,364.458,171.403,47.566,159.298
C01626=1026.369,333.048,364.493,171.398,47.567,159.298
C01627=1026.362,332.800,364.529,171.392,47.567,159.297
C01628=1026.355,332.553,364.565,171.386,47.568,159.296
C01629=1026.348,332.305,364.600,171.380,47.568,159.296
C01630=1026.340,332.058,364.636,171.374,47.568,159.295
C01631=1026.333,331.811,364.671,171.368,47.569,159.294
C01632=1026.325,331.563,364.707,171.362,47.570,159.294
C01633=1026.318,331.316,364.742,171.357,47.570,159.293
C01634=1026.311,331.069,364.778,171.351,47.570,159.292
C01635=1026.304,330.821,364.813,171.344,47.570,159.291
C01636=1026.296,330.573,364.849,171.339,47.571,159.291
C01637=1026.289,330.327,364.884,171.333,47.571,159.290
C01638=1026.281,330.079,364.920,171.328,47.572,159.290
C01639=1026.274,329.831,364.955,171.322,47.572,159.289
C01640=1026.267,329.585,364.991,171.316,47.573,159.288
C01641=1026.260,329.336,365.026,171.310,47.573,159.288
C01642=1026.253,329.089,365.061,171.305,47.574,159.287
C01643=1026.245,328.843,365.097,171.299,47.574,159.286
C01644=1026.238,328.595,365.132,171.292,47.575,159.286
C01645=1026.231,328.347,365.167,171.287,47.575,159.285
C01646=1026.225,328.100,365.202,171.281,47.576,159.284
C01647=1026.216,327.852,365.237,171.276,47.576,159.284
C01648=1026.210,327.605,365.272,171.270,47.577,159.283
C01649=1026.203,327.358,365.308,171.265,47.577,159.282
C01650=1026.195,327.110,365.344,171.258,47.578,159.282
C01651=1026.188,326.863,365.378,171.253,47.579,159.281
C01652=1026.181,326.615,365.412,171.247,47.579,159.281
C01653=1026.173,326.367,365.448,171.242,47.580,159.280
C01654=1026.166,326.120,365.482,171.235,47.581,159.279
C01655=1026.158,325.873,365.517,171.230,47.581,159.279
C01656=1026.151,325.626,365.552,171.224,47.582,159.278
C01657=1026.143,325.378,365.587,171.219,47.583,159.278
C01658=1026.137,325.131,365.622,171.214,47.583,159.277
C01659=1026.129,324.883,365.656,171.207,47.584,159.276
C01660=1026.121,324.635,365.691,171.202,47.585,159.276
C01661=1026.114,324.388,365.726,171.196,47.586,159.275
C01662=1026.107,324.141,365.760,171.191,47.586,159.275
C01663=1026.100,323.893,365.794,171.185,47.587,159.274
C01664=1026.093,323.646,365.829,171.180,47.587,159.274
C01665=1026.085,323.398,365.864,171.174,47.588,159.273
C01666=1026.078,323.150,365.898,171.168,47.589,159.272
C01667=1026.071,322.903,365.933,171.163,47.590,159.272
C01668=1026.063,322.656,365.968,171.158,47.591,159.271
C01669=1026.057,322.433,365.998,171.152,47.592,159.271
C01670=1026.051,322.209,366.030,171.148,47.592,159.270
C01671=1026.044,321.985,366.061,171.142,47.593,159.270
C01672=1026.038,321.762,366.092,171.137,47.594,159.269
C01673=1026.031,321.539,366.123,171.133,47.594,159.269
C01674=1026.025,321.316,366.154,171.127,47.595,159.268
C01675=1026.018,321.092,366.185,171.123,47.596,159.268
C01676=1026.012,320.869,366.217,171.118,47.596,159.267
C01677=1026.004,320.622,366.251,171.112,47.597,159.267
C01678=1025.998,320.374,366.286,171.107,47.598,159.266
C01679=1025.990,320.126,366.319,171.102,47.599,159.266
C01680=1025.983,319.879,366.353,171.096,47.600,159.265
C01681=1025.976,319.631,366.388,171.090,47.601,159.265
C01682=1025.969,319.384,366.422,171.085,47.602,159.264
C01683=1025.962,319.137,366.457,171.079,47.602,159.264
C01684=1025.955,318.889,366.491,171.074,47.603,159.263
C01685=1025.948,318.641,366.525,171.068,47.604,159.263
C01686=1025.941,318.394,366.560,171.063,47.605,159.262
C01687=1025.934,318.146,366.594,171.058,47.606,159.262
C01688=1025.927,317.898,366.628,171.052,47.606,159.261
C01689=1025.919,317.651,366.662,171.047,47.607,159.260
C01690=1025.913,317.403,366.697,171.042,47.609,159.260
C01691=1025.906,317.156,366.730,171.037,47.609,159.260
C01692=1025.899,316.909,366.764,171.031,47.610,159.259
C01693=1025.892,316.661,366.799,171.026,47.611,159.259
C01694=1025.885,316.414,366.833,171.021,47.612,159.258
C01695=1025.878,316.166,366.867,171.015,47.613,159.258
C01696=1025.872,315.918,366.901,171.010,47.614,159.257
C01697=1025.864,315.670,366.935,171.005,47.615,159.257
C01698=1025.857,315.424,366.969,170.999,47.616,159.256
C01699=1025.851,315.176,367.004,170.994,47.617,159.256
C01700=1025.844,314.928,367.038,170.989,47.618,159.255
C01701=1025.837,314.681,367.071,170.984,47.619,159.255
C01702=1025.830,314.433,367.106,170.978,47.620,159.254
C01703=1025.823,314.186,367.139,170.973,47.620,159.254
C01704=1025.816,313.938,367.173,170.968,47.622,159.253
C01705=1025.810,313.690,367.207,170.963,47.623,159.253
C01706=1025.803,313.442,367.241,170.957,47.623,159.252
C01707=1025.796,313.195,367.275,170.952,47.625,159.252
C01708=1025.789,312.948,367.309,170.947,47.626,159.251
C01709=1025.782,312.700,367.343,170.942,47.626,159.251
C01710=1025.776,312.453,367.376,170.936,47.628,159.251
C01711=1025.769,312.205,367.410,170.931,47.629,159.250
C01712=1025.762,311.957,367.445,170.926,47.630,159.250
C01713=1025.756,311.710,367.478,170.921,47.631,159.249
C01714=1025.748,311.462,367.512,170.916,47.632,159.249
C01715=1025.742,311.214,367.546,170.910,47.633,159.248
C01716=1025.736,310.967,367.579,170.905,47.634,159.248
C01717=1025.728,310.719,367.613,170.900,47.635,159.247
C01718=1025.722,310.472,367.646,170.895,47.637,159.247
C01719=1025.715,310.225,367.680,170.890,47.638,159.246
C01720=1025.707,309.977,367.713,170.884,47.639,159.246
C01721=1025.700,309.730,367.746,170.879,47.641,159.246
C01722=1025.693,309.481,367.779,170.874,47.641,159.245
C01723=1025.685,309.234,367.813,170.869,47.643,159.245
C01724=1025.679,308.986,367.845,170.864,47.644,159.245
C01725=1025.672,308.739,367.879,170.859,47.646,159.244
C01726=1025.664,308.491,367.912,170.854,47.646,159.244
C01727=1025.658,308.244,367.945,170.849,47.648,159.243
C01728=1025.651,307.995,367.978,170.844,47.649,159.243
C01729=1025.644,307.774,368.007,170.840,47.650,159.243
C01730=1025.638,307.554,368.037,170.834,47.652,159.242
C01731=1025.632,307.333,368.066,170.830,47.653,159.242
C01732=1025.625,307.112,368.096,170.825,47.654,159.242
C01733=1025.620,306.892,368.125,170.821,47.655,159.241
C01734=1025.614,306.671,368.155,170.817,47.656,159.241
C01735=1025.607,306.450,368.184,170.812,47.658,159.241
C01736=1025.601,306.229,368.213,170.808,47.659,159.240
C01737=1025.594,305.982,368.246,170.803,47.660,159.240
C01738=1025.587,305.734,368.279,170.798,47.662,159.240
C01739=1025.580,305.486,368.312,170.793,47.663,159.239
C01740=1025.573,305.239,368.345,170.788,47.665,159.239
C01741=1025.566,304.991,368.378,170.783,47.666,159.239
C01742=1025.560,304.743,368.411,170.778,47.667,159.238
C01743=1025.552,304.495,368.444,170.773,47.669,159.238
C01744=1025.546,304.248,368.476,170.768,47.670,159.238
C01745=1025.539,304.000,368.510,170.763,47.672,159.237
C01746=1025.532,303.753,368.542,170.758,47.673,159.237
C01747=1025.525,303.504,368.575,170.753,47.675,159.237
C01748=1025.518,303.257,368.608,170.747,47.676,159.236
C01749=1025.511,303.009,368.641,170.743,47.677,159.236
C01750=1025.505,302.761,368.673,170.738,47.679,159.236
C01751=1025.498,302.514,368.706,170.733,47.680,159.235
C01752=1025.491,302.266,368.739,170.728,47.681,159.235
C01753=1025.484,302.018,368.771,170.723,47.683,159.235
C01754=1025.477,301.770,368.804,170.718,47.684,159.234
C01755=1025.470,301.523,368.837,170.713,47.686,159.234
C01756=1025.464,301.276,368.870,170.708,47.687,159.234
C01757=1025.457,301.027,368.903,170.703,47.689,159.233
C01758=1025.450,300.780,368.935,170.699,47.690,159.233
C01759=1025.444,300.532,368.967,170.694,47.692,159.233
C01760=1025.437,300.283,369.000,170.689,47.693,159.232
C01761=1025.430,300.036,369.033,170.684,47.695,159.232
C01762=1025.424,299.789,369.065,170.679,47.696,159.232
C01763=1025.417,299.541,369.098,170.674,47.698,159.231
C01764=1025.410,299.293,369.131,170.669,47.699,159.231
C01765=1025.403,299.045,369.163,170.665,47.701,159.231
C01766=1025.396,298.798,369.196,170.660,47.702,159.231
C01767=1025.390,298.551,369.228,170.655,47.704,159.230
C01768=1025.384,298.302,369.261,170.650,47.705,159.230
C01769=1025.376,298.054,369.293,170.646,47.707,159.230
C01770=1025.370,297.807,369.326,170.641,47.709,159.229
C01771=1025.364,297.559,369.358,170.636,47.710,159.229
C01772=1025.356,297.311,369.391,170.631,47.711,159.229
C01773=1025.350,297.063,369.423,170.627,47.713,159.229
C01774=1025.344,296.815,369.456,170.622,47.715,159.228
C01775=1025.337,296.568,369.488,170.617,47.716,159.228
C01776=1025.331,296.320,369.520,170.612,47.718,159.228
C01777=1025.324,296.073,369.552,170.608,47.719,159.227
C01778=1025.317,295.824,369.585,170.603,47.721,159.227
C01779=1025.311,295.577,369.618,170.598,47.723,159.227
C01780=1025.304,295.329,369.649,170.593,47.724,159.227
C01781=1025.298,295.081,369.682,170.588,47.726,159.226
C01782=1025.291,294.834,369.715,170.584,47.728,159.226
C01783=1025.285,294.586,369.746,170.579,47.729,159.226
C01784=1025.278,294.338,369.779,170.575,47.731,159.226
C01785=1025.272,294.090,369.810,170.570,47.733,159.225
C01786=1025.265,293.842,369.843,170.565,47.735,159.225
C01787=1025.258,293.594,369.875,170.561,47.736,159.225
C01788=1025.251,293.347,369.907,170.556,47.738,159.225
C01789=1025.246,293.135,369.934,170.552,47.739,159.224
C01790=1025.240,292.922,369.961,170.548,47.741,159.224
C01791=1025.234,292.710,369.988,170.543,47.742,159.224
C01792=1025.228,292.498,370.016,170.540,47.744,159.224
C01793=1025.223,292.286,370.044,170.536,47.745,159.223
C01794=1025.217,292.074,370.071,170.532,47.747,159.223
C01795=1025.211,291.862,370.098,170.528,47.748,159.223
C01796=1025.206,291.650,370.125,170.524,47.750,159.223
C01797=1025.200,291.401,370.157,170.519,47.752,159.223
C01798=1025.193,291.154,370.188,170.514,47.753,159.222
C01799=1025.186,290.906,370.221,170.510,47.755,159.222
C01800=1025.179,290.658,370.252,170.506,47.757,159.222
C01801=1025.172,290.410,370.284,170.501,47.759,159.222
C01802=1025.165,290.162,370.315,170.496,47.761,159.222
C01803=1025.158,289.914,370.347,170.491,47.763,159.222
C01804=1025.152,289.666,370.379,170.487,47.765,159.221
C01805=1025.145,289.418,370.411,170.483,47.766,159.221
C01806=1025.139,289.171,370.442,170.478,47.768,159.221
C01807=1025.132,288.923,370.474,170.473,47.770,159.221
C01808=1025.125,288.675,370.505,170.468,47.772,159.221
C01809=1025.119,288.427,370.537,170.464,47.774,159.220
